LIN {X 0,Y 467.673,Z 382.231,A -85,B 0,C 180,E1 -7731.357,E2 -7731.357} C_VEL
LIN {X 0,Y 467.733,Z 382.223,A -85,B 0,C 180,E1 -7733.963,E2 -7733.963} C_VEL
LIN {X 0,Y 467.851,Z 382.207,A -85,B 0,C 180,E1 -7737.417,E2 -7737.417} C_VEL
LIN {X 0,Y 467.873,Z 382.205,A -85,B 0,C 180,E1 -7740,E2 -7740} C_VEL
LIN {X 0,Y 467.851,Z 382.211,A -85,B 0,C 180,E1 -7742.583,E2 -7742.583} C_VEL
LIN {X 0,Y 467.734,Z 382.223,A -85,B 0,C 180,E1 -7746.038,E2 -7746.038} C_VEL
LIN {X 0,Y 467.674,Z 382.232,A -85,B 0,C 180,E1 -7748.643,E2 -7748.643} C_VEL
LIN {X 0,Y 467.648,Z 382.234,A -85,B 0,C 180,E1 -7752.146,E2 -7752.146} C_VEL
LIN {X 0,Y 467.63,Z 382.235,A -85,B 0,C 180,E1 -7755.695,E2 -7755.695} C_VEL
LIN {X 0,Y 467.609,Z 382.239,A -85,B 0,C 180,E1 -7758.765,E2 -7758.765} C_VEL
LIN {X 0,Y 467.573,Z 382.243,A -85,B 0,C 180,E1 -7761.269,E2 -7761.269} C_VEL
LIN {X 0,Y 467.566,Z 382.246,A -85,B 0,C 180,E1 -7763.944,E2 -7763.944} C_VEL
LIN {X 0,Y 467.621,Z 382.239,A -85,B 0,C 180,E1 -7766.8,E2 -7766.8} C_VEL
LIN {X 0,Y 467.547,Z 382.247,A -85,B 0,C 180,E1 -7769.739,E2 -7769.739} C_VEL
LIN {X 0,Y 467.577,Z 382.243,A -85,B 0,C 180,E1 -7772.759,E2 -7772.759} C_VEL
LIN {X 0,Y 467.552,Z 382.247,A -85,B 0,C 180,E1 -7775.89,E2 -7775.89} C_VEL
LIN {X 0,Y 467.614,Z 382.238,A -85,B 0,C 180,E1 -7779.142,E2 -7779.142} C_VEL
LIN {X 0,Y 467.582,Z 382.243,A -85,B 0,C 180,E1 -7782.568,E2 -7782.568} C_VEL
LIN {X 0,Y 467.566,Z 382.243,A -85,B 0,C 180,E1 -7785.054,E2 -7785.054} C_VEL
LIN {X 0,Y 467.586,Z 382.241,A -85,B 0,C 180,E1 -7787.441,E2 -7787.441} C_VEL
LIN {X 0,Y 467.58,Z 382.242,A -85,B 0,C 180,E1 -7790.856,E2 -7790.856} C_VEL
LIN {X 0,Y 467.561,Z 382.246,A -85,B 0,C 180,E1 -7794.261,E2 -7794.261} C_VEL
LIN {X 0,Y 467.581,Z 382.242,A -85,B 0,C 180,E1 -7797.322,E2 -7797.322} C_VEL
LIN {X 0,Y 467.57,Z 382.243,A -85,B 0,C 180,E1 -7800.668,E2 -7800.668} C_VEL
LIN {X 0,Y 467.617,Z 382.236,A -85,B 0,C 180,E1 -7803.201,E2 -7803.201} C_VEL
LIN {X 0,Y 467.595,Z 382.241,A -85,B 0,C 180,E1 -7806.469,E2 -7806.469} C_VEL
LIN {X 0,Y 467.625,Z 382.238,A -85,B 0,C 180,E1 -7809.778,E2 -7809.778} C_VEL
LIN {X 0,Y 467.609,Z 382.238,A -85,B 0,C 180,E1 -7812.507,E2 -7812.507} C_VEL
LIN {X 0,Y 467.6,Z 382.238,A -85,B 0,C 180,E1 -7815.427,E2 -7815.427} C_VEL
LIN {X 0,Y 466.93,Z 382.324,A -85,B 0,C 180,E1 -7816.146,E2 -7816.146} C_VEL
LIN {X 0,Y 464.086,Z 382.678,A -85,B 0,C 180,E1 -7817.315,E2 -7817.315} C_VEL
LIN {X 0,Y 461.687,Z 382.976,A -85,B 0,C 180,E1 -7818.257,E2 -7818.257} C_VEL
LIN {X 0,Y 460.66,Z 383.103,A -85,B 0,C 180,E1 -7818.984,E2 -7818.984} C_VEL
LIN {X 0,Y 460.578,Z 383.114,A -85,B 0,C 180,E1 -7819.231,E2 -7819.231} C_VEL
LIN {X 0,Y 460.724,Z 383.095,A -85,B 0,C 180,E1 -7822.539,E2 -7822.539} C_VEL
LIN {X 0,Y 460.701,Z 383.098,A -85,B 0,C 180,E1 -7824.749,E2 -7824.749} C_VEL
LIN {X 0,Y 460.642,Z 383.109,A -85,B 0,C 180,E1 -7828.252,E2 -7828.252} C_VEL
LIN {X 0,Y 460.422,Z 383.137,A -85,B 0,C 180,E1 -7830,E2 -7830} C_VEL
LIN {X 0,Y 460.136,Z 383.537,A -85,B 0,C 180,E1 -7830.875,E2 -7830.875} C_VEL
LIN {X 0,Y 460.101,Z 387.168,A -85,B 0,C 180,E1 -7834.38,E2 -7834.38} C_VEL
LIN {X 0,Y 460.05,Z 389.931,A -85,B 0,C 180,E1 -7837.02,E2 -7837.02} C_VEL
LIN {X 0,Y 459.887,Z 393.714,A -85,B 0,C 180,E1 -7840.567,E2 -7840.567} C_VEL
LIN {X 0,Y 459.817,Z 396.601,A -85,B 0,C 180,E1 -7843.254,E2 -7843.254} C_VEL
LIN {X 0,Y 459.747,Z 400.031,A -85,B 0,C 180,E1 -7846.427,E2 -7846.427} C_VEL
LIN {X 0,Y 459.761,Z 400.289,A -85,B 0,C 180,E1 -7846.484,E2 -7846.484} C_VEL
LIN {X 0,Y 463,Z 413.86,A -85,B 0,C 180,E1 -7847.018,E2 -7847.018} C_VEL
LIN {X 0,Y 463.452,Z 417.522,A -85,B 0,C 180,E1 -7847.183,E2 -7847.183} C_VEL
LIN {X 0,Y 462.965,Z 429.882,A -85,B 0,C 180,E1 -7847.788,E2 -7847.788} C_VEL
LIN {X 0,Y 462.562,Z 440.759,A -85,B 0,C 180,E1 -7848.492,E2 -7848.492} C_VEL
LIN {X 0,Y 462.154,Z 450.981,A -85,B 0,C 180,E1 -7849.322,E2 -7849.322} C_VEL
LIN {X 0,Y 461.626,Z 460.435,A -85,B 0,C 180,E1 -7850.264,E2 -7850.264} C_VEL
LIN {X 0,Y 461.106,Z 470.133,A -85,B 0,C 180,E1 -7851.457,E2 -7851.457} C_VEL
LIN {X 0,Y 460.671,Z 478.078,A -85,B 0,C 180,E1 -7852.657,E2 -7852.657} C_VEL
LIN {X 0,Y 460.337,Z 485.075,A -85,B 0,C 180,E1 -7853.959,E2 -7853.959} C_VEL
LIN {X 0,Y 460.054,Z 490.904,A -85,B 0,C 180,E1 -7855.324,E2 -7855.324} C_VEL
LIN {X 0,Y 459.888,Z 495.753,A -85,B 0,C 180,E1 -7856.796,E2 -7856.796} C_VEL
LIN {X 0,Y 459.702,Z 499.35,A -85,B 0,C 180,E1 -7858.29,E2 -7858.29} C_VEL
LIN {X 0,Y 459.602,Z 501.158,A -85,B 0,C 180,E1 -7859.353,E2 -7859.353} C_VEL
LIN {X 0,Y 459.552,Z 502.793,A -85,B 0,C 180,E1 -7861.083,E2 -7861.083} C_VEL
LIN {X 0,Y 459.542,Z 502.954,A -85,B 0,C 180,E1 -7862.739,E2 -7862.739} C_VEL
LIN {X 0,Y 459.603,Z 501.586,A -85,B 0,C 180,E1 -7864.456,E2 -7864.456} C_VEL
LIN {X 0,Y 459.699,Z 499.308,A -85,B 0,C 180,E1 -7865.876,E2 -7865.876} C_VEL
LIN {X 0,Y 459.896,Z 495.681,A -85,B 0,C 180,E1 -7867.377,E2 -7867.377} C_VEL
LIN {X 0,Y 460.107,Z 490.878,A -85,B 0,C 180,E1 -7868.829,E2 -7868.829} C_VEL
LIN {X 0,Y 460.383,Z 484.757,A -85,B 0,C 180,E1 -7870.245,E2 -7870.245} C_VEL
LIN {X 0,Y 460.797,Z 477.118,A -85,B 0,C 180,E1 -7871.639,E2 -7871.639} C_VEL
LIN {X 0,Y 461.249,Z 468.89,A -85,B 0,C 180,E1 -7872.85,E2 -7872.85} C_VEL
LIN {X 0,Y 461.723,Z 459.558,A -85,B 0,C 180,E1 -7873.966,E2 -7873.966} C_VEL
LIN {X 0,Y 462.231,Z 448.885,A -85,B 0,C 180,E1 -7874.991,E2 -7874.991} C_VEL
LIN {X 0,Y 462.725,Z 437.513,A -85,B 0,C 180,E1 -7875.863,E2 -7875.863} C_VEL
LIN {X 0,Y 463.176,Z 425.311,A -85,B 0,C 180,E1 -7876.58,E2 -7876.58} C_VEL
LIN {X 0,Y 463.459,Z 416.793,A -85,B 0,C 180,E1 -7876.969,E2 -7876.969} C_VEL
LIN {X 0,Y 460.901,Z 405.422,A -85,B 0,C 180,E1 -7877.46,E2 -7877.46} C_VEL
LIN {X 0,Y 459.754,Z 400.767,A -85,B 0,C 180,E1 -7877.639,E2 -7877.639} C_VEL
LIN {X 0,Y 459.777,Z 398.225,A -85,B 0,C 180,E1 -7880.059,E2 -7880.059} C_VEL
LIN {X 0,Y 459.846,Z 394.757,A -85,B 0,C 180,E1 -7883.412,E2 -7883.412} C_VEL
LIN {X 0,Y 459.973,Z 391.444,A -85,B 0,C 180,E1 -7886.629,E2 -7886.629} C_VEL
LIN {X 0,Y 460.058,Z 388.286,A -85,B 0,C 180,E1 -7889.727,E2 -7889.727} C_VEL
LIN {X 0,Y 460.11,Z 385.256,A -85,B 0,C 180,E1 -7892.726,E2 -7892.726} C_VEL
LIN {X 0,Y 460.168,Z 383.268,A -85,B 0,C 180,E1 -7894.682,E2 -7894.682} C_VEL
LIN {X 0,Y 460.464,Z 383.133,A -85,B 0,C 180,E1 -7897.569,E2 -7897.569} C_VEL
LIN {X 0,Y 460.565,Z 383.117,A -85,B 0,C 180,E1 -7900.384,E2 -7900.384} C_VEL
LIN {X 0,Y 460.56,Z 383.118,A -85,B 0,C 180,E1 -7903.146,E2 -7903.146} C_VEL
LIN {X 0,Y 460.549,Z 383.121,A -85,B 0,C 180,E1 -7905.868,E2 -7905.868} C_VEL
LIN {X 0,Y 460.607,Z 383.111,A -85,B 0,C 180,E1 -7908.559,E2 -7908.559} C_VEL
LIN {X 0,Y 460.689,Z 383.1,A -85,B 0,C 180,E1 -7912.108,E2 -7912.108} C_VEL
LIN {X 0,Y 460.691,Z 383.099,A -85,B 0,C 180,E1 -7914.748,E2 -7914.748} C_VEL
LIN {X 0,Y 460.819,Z 383.082,A -85,B 0,C 180,E1 -7917.378,E2 -7917.378} C_VEL
LIN {X 0,Y 460.846,Z 383.08,A -85,B 0,C 180,E1 -7920,E2 -7920} C_VEL
LIN {X 0,Y 460.818,Z 383.084,A -85,B 0,C 180,E1 -7922.622,E2 -7922.622} C_VEL
LIN {X 0,Y 460.703,Z 383.099,A -85,B 0,C 180,E1 -7926.13,E2 -7926.13} C_VEL
LIN {X 0,Y 460.623,Z 383.11,A -85,B 0,C 180,E1 -7928.776,E2 -7928.776} C_VEL
LIN {X 0,Y 460.607,Z 383.112,A -85,B 0,C 180,E1 -7932.445,E2 -7932.445} C_VEL
LIN {X 0,Y 460.594,Z 383.112,A -85,B 0,C 180,E1 -7935.998,E2 -7935.998} C_VEL
LIN {X 0,Y 460.565,Z 383.114,A -85,B 0,C 180,E1 -7938.902,E2 -7938.902} C_VEL
LIN {X 0,Y 460.51,Z 383.123,A -85,B 0,C 180,E1 -7941.486,E2 -7941.486} C_VEL
LIN {X 0,Y 460.537,Z 383.121,A -85,B 0,C 180,E1 -7944.333,E2 -7944.333} C_VEL
LIN {X 0,Y 460.579,Z 383.116,A -85,B 0,C 180,E1 -7947.243,E2 -7947.243} C_VEL
LIN {X 0,Y 460.505,Z 383.125,A -85,B 0,C 180,E1 -7950.24,E2 -7950.24} C_VEL
LIN {X 0,Y 460.515,Z 383.125,A -85,B 0,C 180,E1 -7953.326,E2 -7953.326} C_VEL
LIN {X 0,Y 460.473,Z 383.132,A -85,B 0,C 180,E1 -7956.53,E2 -7956.53} C_VEL
LIN {X 0,Y 460.575,Z 383.117,A -85,B 0,C 180,E1 -7959.858,E2 -7959.858} C_VEL
LIN {X 0,Y 460.51,Z 383.124,A -85,B 0,C 180,E1 -7962.901,E2 -7962.901} C_VEL
LIN {X 0,Y 460.509,Z 383.125,A -85,B 0,C 180,E1 -7965.831,E2 -7965.831} C_VEL
LIN {X 0,Y 460.581,Z 383.262,A -85,B 0,C 180,E1 -7968.847,E2 -7968.847} C_VEL
LIN {X 0,Y 461.978,Z 390.924,A -85,B 0,C 180,E1 -7972.519,E2 -7972.519} C_VEL
LIN {X 0,Y 462.403,Z 394.851,A -85,B 0,C 180,E1 -7974.202,E2 -7974.202} C_VEL
LIN {X 0,Y 462.054,Z 401.187,A -85,B 0,C 180,E1 -7976.8,E2 -7976.8} C_VEL
LIN {X 0,Y 461.502,Z 410.096,A -85,B 0,C 180,E1 -7980.23,E2 -7980.23} C_VEL
LIN {X 0,Y 461.151,Z 418.397,A -85,B 0,C 180,E1 -7983.283,E2 -7983.283} C_VEL
LIN {X 0,Y 460.78,Z 427.79,A -85,B 0,C 180,E1 -7986.637,E2 -7986.637} C_VEL
LIN {X 0,Y 460.497,Z 437.508,A -85,B 0,C 180,E1 -7989.917,E2 -7989.917} C_VEL
LIN {X 0,Y 460.237,Z 445.764,A -85,B 0,C 180,E1 -7992.676,E2 -7992.676} C_VEL
LIN {X 0,Y 460.163,Z 450.69,A -85,B 0,C 180,E1 -7994.339,E2 -7994.339} C_VEL
LIN {X 0,Y 462.544,Z 465.256,A -85,B 0,C 180,E1 -7994.813,E2 -7994.813} C_VEL
LIN {X 0,Y 463.237,Z 471.072,A -85,B 0,C 180,E1 -7995.054,E2 -7995.054} C_VEL
LIN {X 0,Y 462.854,Z 482.753,A -85,B 0,C 180,E1 -7995.603,E2 -7995.603} C_VEL
LIN {X 0,Y 462.294,Z 495.103,A -85,B 0,C 180,E1 -7996.371,E2 -7996.371} C_VEL
LIN {X 0,Y 461.859,Z 505.182,A -85,B 0,C 180,E1 -7997.168,E2 -7997.168} C_VEL
LIN {X 0,Y 461.401,Z 515.131,A -85,B 0,C 180,E1 -7998.134,E2 -7998.134} C_VEL
LIN {X 0,Y 460.835,Z 524.354,A -85,B 0,C 180,E1 -7999.233,E2 -7999.233} C_VEL
LIN {X 0,Y 460.396,Z 533.354,A -85,B 0,C 180,E1 -8000.555,E2 -8000.555} C_VEL
LIN {X 0,Y 460.054,Z 540.602,A -85,B 0,C 180,E1 -8001.876,E2 -8001.876} C_VEL
LIN {X 0,Y 459.848,Z 545.496,A -85,B 0,C 180,E1 -8002.977,E2 -8002.977} C_VEL
LIN {X 0,Y 459.756,Z 550.26,A -85,B 0,C 180,E1 -8004.297,E2 -8004.297} C_VEL
LIN {X 0,Y 459.58,Z 553.894,A -85,B 0,C 180,E1 -8005.615,E2 -8005.615} C_VEL
LIN {X 0,Y 459.591,Z 555.773,A -85,B 0,C 180,E1 -8006.493,E2 -8006.493} C_VEL
LIN {X 0,Y 459.57,Z 557.175,A -85,B 0,C 180,E1 -8007.37,E2 -8007.37} C_VEL
LIN {X 0,Y 459.494,Z 558.779,A -85,B 0,C 180,E1 -8009.123,E2 -8009.123} C_VEL
LIN {X 0,Y 459.474,Z 558.994,A -85,B 0,C 180,E1 -8010,E2 -8010} C_VEL
LIN {X 0,Y 459.494,Z 558.779,A -85,B 0,C 180,E1 -8010.876,E2 -8010.876} C_VEL
LIN {X 0,Y 459.57,Z 557.179,A -85,B 0,C 180,E1 -8012.629,E2 -8012.629} C_VEL
LIN {X 0,Y 459.591,Z 555.777,A -85,B 0,C 180,E1 -8013.507,E2 -8013.507} C_VEL
LIN {X 0,Y 459.634,Z 552.819,A -85,B 0,C 180,E1 -8014.824,E2 -8014.824} C_VEL
LIN {X 0,Y 459.757,Z 548.818,A -85,B 0,C 180,E1 -8016.142,E2 -8016.142} C_VEL
LIN {X 0,Y 459.929,Z 542.664,A -85,B 0,C 180,E1 -8017.683,E2 -8017.683} C_VEL
LIN {X 0,Y 460.287,Z 535.951,A -85,B 0,C 180,E1 -8019.004,E2 -8019.004} C_VEL
LIN {X 0,Y 460.699,Z 527.624,A -85,B 0,C 180,E1 -8020.325,E2 -8020.325} C_VEL
LIN {X 0,Y 461.15,Z 519.095,A -85,B 0,C 180,E1 -8021.427,E2 -8021.427} C_VEL
LIN {X 0,Y 461.664,Z 508.859,A -85,B 0,C 180,E1 -8022.5,E2 -8022.5} C_VEL
LIN {X 0,Y 462.174,Z 496.862,A -85,B 0,C 180,E1 -8023.509,E2 -8023.509} C_VEL
LIN {X 0,Y 462.717,Z 484.815,A -85,B 0,C 180,E1 -8024.289,E2 -8024.289} C_VEL
LIN {X 0,Y 463.22,Z 472.452,A -85,B 0,C 180,E1 -8024.89,E2 -8024.89} C_VEL
LIN {X 0,Y 463.011,Z 468.654,A -85,B 0,C 180,E1 -8025.05,E2 -8025.05} C_VEL
LIN {X 0,Y 460.929,Z 455.877,A -85,B 0,C 180,E1 -8025.515,E2 -8025.515} C_VEL
LIN {X 0,Y 460.169,Z 450.853,A -85,B 0,C 180,E1 -8025.661,E2 -8025.661} C_VEL
LIN {X 0,Y 460.459,Z 440.42,A -85,B 0,C 180,E1 -8029.178,E2 -8029.178} C_VEL
LIN {X 0,Y 460.726,Z 430.867,A -85,B 0,C 180,E1 -8032.417,E2 -8032.417} C_VEL
LIN {X 0,Y 460.993,Z 422.694,A -85,B 0,C 180,E1 -8035.268,E2 -8035.268} C_VEL
LIN {X 0,Y 461.385,Z 414.794,A -85,B 0,C 180,E1 -8038.177,E2 -8038.177} C_VEL
LIN {X 0,Y 461.803,Z 405.886,A -85,B 0,C 180,E1 -8041.543,E2 -8041.543} C_VEL
LIN {X 0,Y 462.222,Z 399.011,A -85,B 0,C 180,E1 -8044.233,E2 -8044.233} C_VEL
LIN {X 0,Y 462.401,Z 393.857,A -85,B 0,C 180,E1 -8046.337,E2 -8046.337} C_VEL
LIN {X 0,Y 461.392,Z 387.782,A -85,B 0,C 180,E1 -8049.028,E2 -8049.028} C_VEL
LIN {X 0,Y 460.548,Z 383.118,A -85,B 0,C 180,E1 -8051.303,E2 -8051.303} C_VEL
LIN {X 0,Y 460.512,Z 383.124,A -85,B 0,C 180,E1 -8054.588,E2 -8054.588} C_VEL
LIN {X 0,Y 460.519,Z 383.122,A -85,B 0,C 180,E1 -8057.818,E2 -8057.818} C_VEL
LIN {X 0,Y 460.562,Z 383.118,A -85,B 0,C 180,E1 -8061.098,E2 -8061.098} C_VEL
LIN {X 0,Y 460.507,Z 383.124,A -85,B 0,C 180,E1 -8064.554,E2 -8064.554} C_VEL
LIN {X 0,Y 460.525,Z 383.119,A -85,B 0,C 180,E1 -8067.715,E2 -8067.715} C_VEL
LIN {X 0,Y 460.532,Z 383.122,A -85,B 0,C 180,E1 -8070.768,E2 -8070.768} C_VEL
LIN {X 0,Y 460.56,Z 383.116,A -85,B 0,C 180,E1 -8073.735,E2 -8073.735} C_VEL
LIN {X 0,Y 460.538,Z 383.121,A -85,B 0,C 180,E1 -8076.624,E2 -8076.624} C_VEL
LIN {X 0,Y 460.544,Z 383.119,A -85,B 0,C 180,E1 -8079.452,E2 -8079.452} C_VEL
LIN {X 0,Y 460.551,Z 383.118,A -85,B 0,C 180,E1 -8082.23,E2 -8082.23} C_VEL
LIN {X 0,Y 460.556,Z 383.119,A -85,B 0,C 180,E1 -8084.965,E2 -8084.965} C_VEL
LIN {X 0,Y 460.604,Z 383.113,A -85,B 0,C 180,E1 -8088.559,E2 -8088.559} C_VEL
LIN {X 0,Y 460.686,Z 383.101,A -85,B 0,C 180,E1 -8092.108,E2 -8092.108} C_VEL
LIN {X 0,Y 460.688,Z 383.103,A -85,B 0,C 180,E1 -8094.748,E2 -8094.748} C_VEL
LIN {X 0,Y 460.816,Z 383.084,A -85,B 0,C 180,E1 -8097.378,E2 -8097.378} C_VEL
LIN {X 0,Y 460.844,Z 383.081,A -85,B 0,C 180,E1 -8100,E2 -8100} C_VEL
LIN {X 0,Y 460.816,Z 383.087,A -85,B 0,C 180,E1 -8102.623,E2 -8102.623} C_VEL
LIN {X 0,Y 460.701,Z 383.1,A -85,B 0,C 180,E1 -8106.13,E2 -8106.13} C_VEL
LIN {X 0,Y 460.621,Z 383.11,A -85,B 0,C 180,E1 -8108.776,E2 -8108.776} C_VEL
LIN {X 0,Y 460.604,Z 383.113,A -85,B 0,C 180,E1 -8112.445,E2 -8112.445} C_VEL
LIN {X 0,Y 460.591,Z 383.113,A -85,B 0,C 180,E1 -8115.998,E2 -8115.998} C_VEL
LIN {X 0,Y 460.563,Z 383.117,A -85,B 0,C 180,E1 -8118.902,E2 -8118.902} C_VEL
LIN {X 0,Y 460.508,Z 383.122,A -85,B 0,C 180,E1 -8121.486,E2 -8121.486} C_VEL
LIN {X 0,Y 460.535,Z 383.121,A -85,B 0,C 180,E1 -8124.333,E2 -8124.333} C_VEL
LIN {X 0,Y 460.577,Z 383.114,A -85,B 0,C 180,E1 -8127.244,E2 -8127.244} C_VEL
LIN {X 0,Y 460.504,Z 383.126,A -85,B 0,C 180,E1 -8130.241,E2 -8130.241} C_VEL
LIN {X 0,Y 460.523,Z 383.12,A -85,B 0,C 180,E1 -8133.326,E2 -8133.326} C_VEL
LIN {X 0,Y 460.475,Z 383.128,A -85,B 0,C 180,E1 -8136.53,E2 -8136.53} C_VEL
LIN {X 0,Y 460.573,Z 383.116,A -85,B 0,C 180,E1 -8139.858,E2 -8139.858} C_VEL
LIN {X 0,Y 460.509,Z 383.122,A -85,B 0,C 180,E1 -8142.901,E2 -8142.901} C_VEL
LIN {X 0,Y 460.508,Z 383.124,A -85,B 0,C 180,E1 -8145.831,E2 -8145.831} C_VEL
LIN {X 0,Y 460.528,Z 383.12,A -85,B 0,C 180,E1 -8148.99,E2 -8148.99} C_VEL
LIN {X 0,Y 460.524,Z 383.12,A -85,B 0,C 180,E1 -8151.268,E2 -8151.268} C_VEL
LIN {X 0,Y 460.511,Z 383.124,A -85,B 0,C 180,E1 -8154.556,E2 -8154.556} C_VEL
LIN {X 0,Y 460.531,Z 383.121,A -85,B 0,C 180,E1 -8157.717,E2 -8157.717} C_VEL
LIN {X 0,Y 460.54,Z 383.118,A -85,B 0,C 180,E1 -8160.77,E2 -8160.77} C_VEL
LIN {X 0,Y 460.564,Z 383.119,A -85,B 0,C 180,E1 -8163.736,E2 -8163.736} C_VEL
LIN {X 0,Y 460.548,Z 383.118,A -85,B 0,C 180,E1 -8166.625,E2 -8166.625} C_VEL
LIN {X 0,Y 460.554,Z 383.119,A -85,B 0,C 180,E1 -8169.454,E2 -8169.454} C_VEL
LIN {X 0,Y 460.56,Z 383.119,A -85,B 0,C 180,E1 -8172.231,E2 -8172.231} C_VEL
LIN {X 0,Y 460.568,Z 383.115,A -85,B 0,C 180,E1 -8174.965,E2 -8174.965} C_VEL
LIN {X 0,Y 460.614,Z 383.11,A -85,B 0,C 180,E1 -8178.56,E2 -8178.56} C_VEL
LIN {X 0,Y 460.578,Z 383.114,A -85,B 0,C 180,E1 -8179.231,E2 -8179.231} C_VEL
LIN {X 0,Y 459.922,Z 383.199,A -85,B 0,C 180,E1 -8179.961,E2 -8179.961} C_VEL
LIN {X 0,Y 457.106,Z 383.549,A -85,B 0,C 180,E1 -8181.147,E2 -8181.147} C_VEL
LIN {X 0,Y 454.729,Z 383.845,A -85,B 0,C 180,E1 -8182.105,E2 -8182.105} C_VEL
LIN {X 0,Y 453.718,Z 383.967,A -85,B 0,C 180,E1 -8182.844,E2 -8182.844} C_VEL
LIN {X 0,Y 453.641,Z 383.976,A -85,B 0,C 180,E1 -8183.094,E2 -8183.094} C_VEL
LIN {X 0,Y 453.675,Z 383.973,A -85,B 0,C 180,E1 -8184.667,E2 -8184.667} C_VEL
LIN {X 0,Y 453.615,Z 383.985,A -85,B 0,C 180,E1 -8188.225,E2 -8188.225} C_VEL
LIN {X 0,Y 453.392,Z 384.013,A -85,B 0,C 180,E1 -8190,E2 -8190} C_VEL
LIN {X 0,Y 453.068,Z 384.308,A -85,B 0,C 180,E1 -8190.889,E2 -8190.889} C_VEL
LIN {X 0,Y 453.038,Z 387.969,A -85,B 0,C 180,E1 -8194.449,E2 -8194.449} C_VEL
LIN {X 0,Y 452.964,Z 390.73,A -85,B 0,C 180,E1 -8197.13,E2 -8197.13} C_VEL
LIN {X 0,Y 452.838,Z 394.587,A -85,B 0,C 180,E1 -8200.733,E2 -8200.733} C_VEL
LIN {X 0,Y 452.733,Z 397.492,A -85,B 0,C 180,E1 -8203.465,E2 -8203.465} C_VEL
LIN {X 0,Y 452.696,Z 400.503,A -85,B 0,C 180,E1 -8206.227,E2 -8206.227} C_VEL
LIN {X 0,Y 456.108,Z 414.964,A -85,B 0,C 180,E1 -8206.817,E2 -8206.817} C_VEL
LIN {X 0,Y 456.603,Z 417.501,A -85,B 0,C 180,E1 -8206.941,E2 -8206.941} C_VEL
LIN {X 0,Y 456.094,Z 430.76,A -85,B 0,C 180,E1 -8207.602,E2 -8207.602} C_VEL
LIN {X 0,Y 455.647,Z 441.569,A -85,B 0,C 180,E1 -8208.316,E2 -8208.316} C_VEL
LIN {X 0,Y 455.136,Z 452.929,A -85,B 0,C 180,E1 -8209.276,E2 -8209.276} C_VEL
LIN {X 0,Y 454.533,Z 463.217,A -85,B 0,C 180,E1 -8210.358,E2 -8210.358} C_VEL
LIN {X 0,Y 454.005,Z 472.929,A -85,B 0,C 180,E1 -8211.635,E2 -8211.635} C_VEL
LIN {X 0,Y 453.499,Z 481.425,A -85,B 0,C 180,E1 -8213.036,E2 -8213.036} C_VEL
LIN {X 0,Y 453.161,Z 488.507,A -85,B 0,C 180,E1 -8214.51,E2 -8214.51} C_VEL
LIN {X 0,Y 452.895,Z 493.503,A -85,B 0,C 180,E1 -8215.836,E2 -8215.836} C_VEL
LIN {X 0,Y 452.794,Z 497.6,A -85,B 0,C 180,E1 -8217.25,E2 -8217.25} C_VEL
LIN {X 0,Y 452.572,Z 500.759,A -85,B 0,C 180,E1 -8218.776,E2 -8218.776} C_VEL
LIN {X 0,Y 452.497,Z 502.208,A -85,B 0,C 180,E1 -8219.802,E2 -8219.802} C_VEL
LIN {X 0,Y 452.461,Z 503.357,A -85,B 0,C 180,E1 -8221.316,E2 -8221.316} C_VEL
LIN {X 0,Y 452.471,Z 503.272,A -85,B 0,C 180,E1 -8222.991,E2 -8222.991} C_VEL
LIN {X 0,Y 452.525,Z 501.894,A -85,B 0,C 180,E1 -8224.601,E2 -8224.601} C_VEL
LIN {X 0,Y 452.661,Z 499.306,A -85,B 0,C 180,E1 -8226.162,E2 -8226.162} C_VEL
LIN {X 0,Y 452.869,Z 495.523,A -85,B 0,C 180,E1 -8227.677,E2 -8227.677} C_VEL
LIN {X 0,Y 453.12,Z 490.496,A -85,B 0,C 180,E1 -8229.148,E2 -8229.148} C_VEL
LIN {X 0,Y 453.472,Z 484.031,A -85,B 0,C 180,E1 -8230.611,E2 -8230.611} C_VEL
LIN {X 0,Y 453.879,Z 476.356,A -85,B 0,C 180,E1 -8231.991,E2 -8231.991} C_VEL
LIN {X 0,Y 454.33,Z 468.446,A -85,B 0,C 180,E1 -8233.139,E2 -8233.139} C_VEL
LIN {X 0,Y 454.873,Z 458.449,A -85,B 0,C 180,E1 -8234.315,E2 -8234.315} C_VEL
LIN {X 0,Y 455.35,Z 448.873,A -85,B 0,C 180,E1 -8235.232,E2 -8235.232} C_VEL
LIN {X 0,Y 455.862,Z 438.031,A -85,B 0,C 180,E1 -8236.071,E2 -8236.071} C_VEL
LIN {X 0,Y 456.32,Z 426.219,A -85,B 0,C 180,E1 -8236.781,E2 -8236.781} C_VEL
LIN {X 0,Y 456.459,Z 416.694,A -85,B 0,C 180,E1 -8237.229,E2 -8237.229} C_VEL
LIN {X 0,Y 453.32,Z 403.86,A -85,B 0,C 180,E1 -8237.78,E2 -8237.78} C_VEL
LIN {X 0,Y 452.684,Z 401.216,A -85,B 0,C 180,E1 -8237.894,E2 -8237.894} C_VEL
LIN {X 0,Y 452.71,Z 398.088,A -85,B 0,C 180,E1 -8240.914,E2 -8240.914} C_VEL
LIN {X 0,Y 452.808,Z 395.044,A -85,B 0,C 180,E1 -8243.857,E2 -8243.857} C_VEL
LIN {X 0,Y 452.929,Z 391.77,A -85,B 0,C 180,E1 -8247.106,E2 -8247.106} C_VEL
LIN {X 0,Y 453.009,Z 388.584,A -85,B 0,C 180,E1 -8250.234,E2 -8250.234} C_VEL
LIN {X 0,Y 453.064,Z 385.546,A -85,B 0,C 180,E1 -8253.266,E2 -8253.266} C_VEL
LIN {X 0,Y 453.127,Z 384.547,A -85,B 0,C 180,E1 -8254.26,E2 -8254.26} C_VEL
LIN {X 0,Y 453.189,Z 384.038,A -85,B 0,C 180,E1 -8255.246,E2 -8255.246} C_VEL
LIN {X 0,Y 453.459,Z 384.006,A -85,B 0,C 180,E1 -8258.163,E2 -8258.163} C_VEL
LIN {X 0,Y 453.517,Z 383.997,A -85,B 0,C 180,E1 -8261.008,E2 -8261.008} C_VEL
LIN {X 0,Y 453.563,Z 383.988,A -85,B 0,C 180,E1 -8263.879,E2 -8263.879} C_VEL
LIN {X 0,Y 453.558,Z 383.99,A -85,B 0,C 180,E1 -8267.471,E2 -8267.471} C_VEL
LIN {X 0,Y 453.587,Z 383.986,A -85,B 0,C 180,E1 -8271.086,E2 -8271.086} C_VEL
LIN {X 0,Y 453.671,Z 383.975,A -85,B 0,C 180,E1 -8273.774,E2 -8273.774} C_VEL
LIN {X 0,Y 453.759,Z 383.962,A -85,B 0,C 180,E1 -8277.337,E2 -8277.337} C_VEL
LIN {X 0,Y 453.816,Z 383.955,A -85,B 0,C 180,E1 -8280,E2 -8280} C_VEL
LIN {X 0,Y 453.759,Z 383.964,A -85,B 0,C 180,E1 -8282.663,E2 -8282.663} C_VEL
LIN {X 0,Y 453.67,Z 383.976,A -85,B 0,C 180,E1 -8286.225,E2 -8286.225} C_VEL
LIN {X 0,Y 453.587,Z 383.987,A -85,B 0,C 180,E1 -8288.913,E2 -8288.913} C_VEL
LIN {X 0,Y 453.557,Z 383.99,A -85,B 0,C 180,E1 -8292.529,E2 -8292.529} C_VEL
LIN {X 0,Y 453.539,Z 383.99,A -85,B 0,C 180,E1 -8296.196,E2 -8296.196} C_VEL
LIN {X 0,Y 453.514,Z 383.992,A -85,B 0,C 180,E1 -8299.041,E2 -8299.041} C_VEL
LIN {X 0,Y 453.471,Z 384.001,A -85,B 0,C 180,E1 -8301.836,E2 -8301.836} C_VEL
LIN {X 0,Y 453.509,Z 383.997,A -85,B 0,C 180,E1 -8304.735,E2 -8304.735} C_VEL
LIN {X 0,Y 453.533,Z 383.994,A -85,B 0,C 180,E1 -8307.961,E2 -8307.961} C_VEL
LIN {X 0,Y 453.46,Z 384.002,A -85,B 0,C 180,E1 -8311.525,E2 -8311.525} C_VEL
LIN {X 0,Y 453.478,Z 384.001,A -85,B 0,C 180,E1 -8314.777,E2 -8314.777} C_VEL
LIN {X 0,Y 453.482,Z 384,A -85,B 0,C 180,E1 -8318.31,E2 -8318.31} C_VEL
LIN {X 0,Y 453.513,Z 383.997,A -85,B 0,C 180,E1 -8320.607,E2 -8320.607} C_VEL
LIN {X 0,Y 453.463,Z 384.002,A -85,B 0,C 180,E1 -8324.221,E2 -8324.221} C_VEL
LIN {X 0,Y 453.461,Z 384.004,A -85,B 0,C 180,E1 -8327.006,E2 -8327.006} C_VEL
LIN {X 0,Y 453.526,Z 384.139,A -85,B 0,C 180,E1 -8328.513,E2 -8328.513} C_VEL
LIN {X 0,Y 454.528,Z 389.726,A -85,B 0,C 180,E1 -8331.25,E2 -8331.25} C_VEL
LIN {X 0,Y 455.317,Z 394.234,A -85,B 0,C 180,E1 -8333.383,E2 -8333.383} C_VEL
LIN {X 0,Y 455.279,Z 398.473,A -85,B 0,C 180,E1 -8335.17,E2 -8335.17} C_VEL
LIN {X 0,Y 454.88,Z 404.896,A -85,B 0,C 180,E1 -8337.787,E2 -8337.787} C_VEL
LIN {X 0,Y 454.363,Z 414.1,A -85,B 0,C 180,E1 -8341.347,E2 -8341.347} C_VEL
LIN {X 0,Y 453.945,Z 422.089,A -85,B 0,C 180,E1 -8344.311,E2 -8344.311} C_VEL
LIN {X 0,Y 453.673,Z 430.213,A -85,B 0,C 180,E1 -8347.215,E2 -8347.215} C_VEL
LIN {X 0,Y 453.409,Z 439.867,A -85,B 0,C 180,E1 -8350.534,E2 -8350.534} C_VEL
LIN {X 0,Y 453.075,Z 450.258,A -85,B 0,C 180,E1 -8354.098,E2 -8354.098} C_VEL
LIN {X 0,Y 455.051,Z 462.267,A -85,B 0,C 180,E1 -8354.475,E2 -8354.475} C_VEL
LIN {X 0,Y 456.336,Z 471.909,A -85,B 0,C 180,E1 -8354.879,E2 -8354.879} C_VEL
LIN {X 0,Y 455.861,Z 484.275,A -85,B 0,C 180,E1 -8355.491,E2 -8355.491} C_VEL
LIN {X 0,Y 455.282,Z 496.181,A -85,B 0,C 180,E1 -8356.271,E2 -8356.271} C_VEL
LIN {X 0,Y 454.791,Z 506.767,A -85,B 0,C 180,E1 -8357.156,E2 -8357.156} C_VEL
LIN {X 0,Y 454.295,Z 516.635,A -85,B 0,C 180,E1 -8358.172,E2 -8358.172} C_VEL
LIN {X 0,Y 453.714,Z 525.536,A -85,B 0,C 180,E1 -8359.288,E2 -8359.288} C_VEL
LIN {X 0,Y 453.299,Z 534.234,A -85,B 0,C 180,E1 -8360.631,E2 -8360.631} C_VEL
LIN {X 0,Y 452.924,Z 541.184,A -85,B 0,C 180,E1 -8361.972,E2 -8361.972} C_VEL
LIN {X 0,Y 452.71,Z 547.416,A -85,B 0,C 180,E1 -8363.493,E2 -8363.493} C_VEL
LIN {X 0,Y 452.567,Z 552.377,A -85,B 0,C 180,E1 -8365.1,E2 -8365.1} C_VEL
LIN {X 0,Y 452.494,Z 555.337,A -85,B 0,C 180,E1 -8366.438,E2 -8366.438} C_VEL
LIN {X 0,Y 452.496,Z 556.749,A -85,B 0,C 180,E1 -8367.329,E2 -8367.329} C_VEL
LIN {X 0,Y 452.433,Z 558.367,A -85,B 0,C 180,E1 -8369.11,E2 -8369.11} C_VEL
LIN {X 0,Y 452.41,Z 558.586,A -85,B 0,C 180,E1 -8370,E2 -8370} C_VEL
LIN {X 0,Y 452.433,Z 558.371,A -85,B 0,C 180,E1 -8370.89,E2 -8370.89} C_VEL
LIN {X 0,Y 452.496,Z 556.759,A -85,B 0,C 180,E1 -8372.67,E2 -8372.67} C_VEL
LIN {X 0,Y 452.493,Z 555.351,A -85,B 0,C 180,E1 -8373.562,E2 -8373.562} C_VEL
LIN {X 0,Y 452.567,Z 552.394,A -85,B 0,C 180,E1 -8374.899,E2 -8374.899} C_VEL
LIN {X 0,Y 452.686,Z 547.533,A -85,B 0,C 180,E1 -8376.481,E2 -8376.481} C_VEL
LIN {X 0,Y 452.926,Z 541.219,A -85,B 0,C 180,E1 -8378.027,E2 -8378.027} C_VEL
LIN {X 0,Y 453.309,Z 534.281,A -85,B 0,C 180,E1 -8379.368,E2 -8379.368} C_VEL
LIN {X 0,Y 453.697,Z 525.596,A -85,B 0,C 180,E1 -8380.712,E2 -8380.712} C_VEL
LIN {X 0,Y 454.277,Z 516.707,A -85,B 0,C 180,E1 -8381.828,E2 -8381.828} C_VEL
LIN {X 0,Y 454.807,Z 506.763,A -85,B 0,C 180,E1 -8382.852,E2 -8382.852} C_VEL
LIN {X 0,Y 455.266,Z 496.288,A -85,B 0,C 180,E1 -8383.729,E2 -8383.729} C_VEL
LIN {X 0,Y 455.803,Z 484.386,A -85,B 0,C 180,E1 -8384.51,E2 -8384.51} C_VEL
LIN {X 0,Y 456.338,Z 472.025,A -85,B 0,C 180,E1 -8385.12,E2 -8385.12} C_VEL
LIN {X 0,Y 454.636,Z 459.724,A -85,B 0,C 180,E1 -8385.622,E2 -8385.622} C_VEL
LIN {X 0,Y 453.075,Z 450.464,A -85,B 0,C 180,E1 -8385.902,E2 -8385.902} C_VEL
LIN {X 0,Y 453.416,Z 440.196,A -85,B 0,C 180,E1 -8389.466,E2 -8389.466} C_VEL
LIN {X 0,Y 453.651,Z 431.951,A -85,B 0,C 180,E1 -8392.305,E2 -8392.305} C_VEL
LIN {X 0,Y 453.951,Z 423.813,A -85,B 0,C 180,E1 -8395.197,E2 -8395.197} C_VEL
LIN {X 0,Y 454.363,Z 415.899,A -85,B 0,C 180,E1 -8398.156,E2 -8398.156} C_VEL
LIN {X 0,Y 454.844,Z 406.396,A -85,B 0,C 180,E1 -8401.806,E2 -8401.806} C_VEL
LIN {X 0,Y 455.256,Z 400.132,A -85,B 0,C 180,E1 -8404.295,E2 -8404.295} C_VEL
LIN {X 0,Y 455.481,Z 396.271,A -85,B 0,C 180,E1 -8405.896,E2 -8405.896} C_VEL
LIN {X 0,Y 454.877,Z 391.457,A -85,B 0,C 180,E1 -8408.004,E2 -8408.004} C_VEL
LIN {X 0,Y 453.518,Z 384.02,A -85,B 0,C 180,E1 -8411.506,E2 -8411.506} C_VEL
LIN {X 0,Y 453.482,Z 383.999,A -85,B 0,C 180,E1 -8414.528,E2 -8414.528} C_VEL
LIN {X 0,Y 453.476,Z 384,A -85,B 0,C 180,E1 -8418.209,E2 -8418.209} C_VEL
LIN {X 0,Y 453.526,Z 383.995,A -85,B 0,C 180,E1 -8420.787,E2 -8420.787} C_VEL
LIN {X 0,Y 453.451,Z 384.001,A -85,B 0,C 180,E1 -8423.917,E2 -8423.917} C_VEL
LIN {X 0,Y 453.476,Z 384.001,A -85,B 0,C 180,E1 -8427.151,E2 -8427.151} C_VEL
LIN {X 0,Y 453.468,Z 383.999,A -85,B 0,C 180,E1 -8430.268,E2 -8430.268} C_VEL
LIN {X 0,Y 453.506,Z 383.996,A -85,B 0,C 180,E1 -8433.294,E2 -8433.294} C_VEL
LIN {X 0,Y 453.495,Z 383.997,A -85,B 0,C 180,E1 -8436.238,E2 -8436.238} C_VEL
LIN {X 0,Y 453.475,Z 384.001,A -85,B 0,C 180,E1 -8439.117,E2 -8439.117} C_VEL
LIN {X 0,Y 453.503,Z 383.995,A -85,B 0,C 180,E1 -8441.944,E2 -8441.944} C_VEL
LIN {X 0,Y 453.53,Z 383.994,A -85,B 0,C 180,E1 -8444.726,E2 -8444.726} C_VEL
LIN {X 0,Y 453.552,Z 383.991,A -85,B 0,C 180,E1 -8448.379,E2 -8448.379} C_VEL
LIN {X 0,Y 453.643,Z 383.978,A -85,B 0,C 180,E1 -8451.985,E2 -8451.985} C_VEL
LIN {X 0,Y 453.662,Z 383.978,A -85,B 0,C 180,E1 -8454.667,E2 -8454.667} C_VEL
LIN {X 0,Y 453.756,Z 383.963,A -85,B 0,C 180,E1 -8457.337,E2 -8457.337} C_VEL
LIN {X 0,Y 453.814,Z 383.957,A -85,B 0,C 180,E1 -8460,E2 -8460} C_VEL
LIN {X 0,Y 453.757,Z 383.967,A -85,B 0,C 180,E1 -8462.663,E2 -8462.663} C_VEL
LIN {X 0,Y 453.668,Z 383.977,A -85,B 0,C 180,E1 -8466.226,E2 -8466.226} C_VEL
LIN {X 0,Y 453.585,Z 383.987,A -85,B 0,C 180,E1 -8468.914,E2 -8468.914} C_VEL
LIN {X 0,Y 453.554,Z 383.992,A -85,B 0,C 180,E1 -8472.529,E2 -8472.529} C_VEL
LIN {X 0,Y 453.536,Z 383.994,A -85,B 0,C 180,E1 -8476.196,E2 -8476.196} C_VEL
LIN {X 0,Y 453.512,Z 383.995,A -85,B 0,C 180,E1 -8479.041,E2 -8479.041} C_VEL
LIN {X 0,Y 453.469,Z 384.001,A -85,B 0,C 180,E1 -8481.837,E2 -8481.837} C_VEL
LIN {X 0,Y 453.507,Z 383.996,A -85,B 0,C 180,E1 -8484.735,E2 -8484.735} C_VEL
LIN {X 0,Y 453.53,Z 383.993,A -85,B 0,C 180,E1 -8487.962,E2 -8487.962} C_VEL
LIN {X 0,Y 453.46,Z 384,A -85,B 0,C 180,E1 -8491.526,E2 -8491.526} C_VEL
LIN {X 0,Y 453.484,Z 383.998,A -85,B 0,C 180,E1 -8494.779,E2 -8494.779} C_VEL
LIN {X 0,Y 453.481,Z 384,A -85,B 0,C 180,E1 -8498.31,E2 -8498.31} C_VEL
LIN {X 0,Y 453.511,Z 383.995,A -85,B 0,C 180,E1 -8500.607,E2 -8500.607} C_VEL
LIN {X 0,Y 453.462,Z 384.002,A -85,B 0,C 180,E1 -8504.222,E2 -8504.222} C_VEL
LIN {X 0,Y 453.46,Z 384,A -85,B 0,C 180,E1 -8507.006,E2 -8507.006} C_VEL
LIN {X 0,Y 453.515,Z 383.994,A -85,B 0,C 180,E1 -8510.554,E2 -8510.554} C_VEL
LIN {X 0,Y 453.455,Z 384.003,A -85,B 0,C 180,E1 -8513.918,E2 -8513.918} C_VEL
LIN {X 0,Y 453.482,Z 383.997,A -85,B 0,C 180,E1 -8517.152,E2 -8517.152} C_VEL
LIN {X 0,Y 453.475,Z 384.001,A -85,B 0,C 180,E1 -8520.269,E2 -8520.269} C_VEL
LIN {X 0,Y 453.507,Z 383.994,A -85,B 0,C 180,E1 -8523.295,E2 -8523.295} C_VEL
LIN {X 0,Y 453.505,Z 383.996,A -85,B 0,C 180,E1 -8526.24,E2 -8526.24} C_VEL
LIN {X 0,Y 453.485,Z 383.997,A -85,B 0,C 180,E1 -8529.118,E2 -8529.118} C_VEL
LIN {X 0,Y 453.513,Z 383.996,A -85,B 0,C 180,E1 -8531.945,E2 -8531.945} C_VEL
LIN {X 0,Y 453.543,Z 383.99,A -85,B 0,C 180,E1 -8534.727,E2 -8534.727} C_VEL
LIN {X 0,Y 453.563,Z 383.988,A -85,B 0,C 180,E1 -8538.38,E2 -8538.38} C_VEL
LIN {X 0,Y 453.656,Z 383.978,A -85,B 0,C 180,E1 -8541.986,E2 -8541.986} C_VEL
LIN {X 0,Y 453.641,Z 383.976,A -85,B 0,C 180,E1 -8543.094,E2 -8543.094} C_VEL
LIN {X 0,Y 452.95,Z 384.066,A -85,B 0,C 180,E1 -8543.834,E2 -8543.834} C_VEL
LIN {X 0,Y 449.968,Z 384.436,A -85,B 0,C 180,E1 -8545.035,E2 -8545.035} C_VEL
LIN {X 0,Y 447.492,Z 384.745,A -85,B 0,C 180,E1 -8546.004,E2 -8546.004} C_VEL
LIN {X 0,Y 446.501,Z 384.867,A -85,B 0,C 180,E1 -8546.755,E2 -8546.755} C_VEL
LIN {X 0,Y 446.46,Z 384.872,A -85,B 0,C 180,E1 -8547.008,E2 -8547.008} C_VEL
LIN {X 0,Y 446.505,Z 384.87,A -85,B 0,C 180,E1 -8549.098,E2 -8549.098} C_VEL
LIN {X 0,Y 446.002,Z 385.094,A -85,B 0,C 180,E1 -8550.903,E2 -8550.903} C_VEL
LIN {X 0,Y 445.977,Z 388.79,A -85,B 0,C 180,E1 -8554.519,E2 -8554.519} C_VEL
LIN {X 0,Y 445.904,Z 391.595,A -85,B 0,C 180,E1 -8557.244,E2 -8557.244} C_VEL
LIN {X 0,Y 445.775,Z 395.504,A -85,B 0,C 180,E1 -8560.905,E2 -8560.905} C_VEL
LIN {X 0,Y 445.675,Z 398.424,A -85,B 0,C 180,E1 -8563.682,E2 -8563.682} C_VEL
LIN {X 0,Y 445.631,Z 400.926,A -85,B 0,C 180,E1 -8565.983,E2 -8565.983} C_VEL
LIN {X 0,Y 448.832,Z 414.31,A -85,B 0,C 180,E1 -8566.528,E2 -8566.528} C_VEL
LIN {X 0,Y 449.721,Z 418.364,A -85,B 0,C 180,E1 -8566.73,E2 -8566.73} C_VEL
LIN {X 0,Y 449.237,Z 431.256,A -85,B 0,C 180,E1 -8567.387,E2 -8567.387} C_VEL
LIN {X 0,Y 448.759,Z 442.19,A -85,B 0,C 180,E1 -8568.123,E2 -8568.123} C_VEL
LIN {X 0,Y 448.208,Z 453.596,A -85,B 0,C 180,E1 -8569.106,E2 -8569.106} C_VEL
LIN {X 0,Y 447.583,Z 463.877,A -85,B 0,C 180,E1 -8570.209,E2 -8570.209} C_VEL
LIN {X 0,Y 447.03,Z 472.828,A -85,B 0,C 180,E1 -8571.396,E2 -8571.396} C_VEL
LIN {X 0,Y 446.587,Z 480.652,A -85,B 0,C 180,E1 -8572.678,E2 -8572.678} C_VEL
LIN {X 0,Y 446.155,Z 487.987,A -85,B 0,C 180,E1 -8574.177,E2 -8574.177} C_VEL
LIN {X 0,Y 445.87,Z 493.489,A -85,B 0,C 180,E1 -8575.609,E2 -8575.609} C_VEL
LIN {X 0,Y 445.719,Z 498.103,A -85,B 0,C 180,E1 -8577.21,E2 -8577.21} C_VEL
LIN {X 0,Y 445.555,Z 500.336,A -85,B 0,C 180,E1 -8578.242,E2 -8578.242} C_VEL
LIN {X 0,Y 445.412,Z 502.667,A -85,B 0,C 180,E1 -8579.792,E2 -8579.792} C_VEL
LIN {X 0,Y 445.366,Z 503.845,A -85,B 0,C 180,E1 -8581.555,E2 -8581.555} C_VEL
LIN {X 0,Y 445.391,Z 503.587,A -85,B 0,C 180,E1 -8583.247,E2 -8583.247} C_VEL
LIN {X 0,Y 445.49,Z 502.044,A -85,B 0,C 180,E1 -8584.88,E2 -8584.88} C_VEL
LIN {X 0,Y 445.622,Z 499.279,A -85,B 0,C 180,E1 -8586.454,E2 -8586.454} C_VEL
LIN {X 0,Y 445.842,Z 495.302,A -85,B 0,C 180,E1 -8587.985,E2 -8587.985} C_VEL
LIN {X 0,Y 446.142,Z 490.099,A -85,B 0,C 180,E1 -8589.476,E2 -8589.476} C_VEL
LIN {X 0,Y 446.504,Z 483.6,A -85,B 0,C 180,E1 -8590.929,E2 -8590.929} C_VEL
LIN {X 0,Y 446.956,Z 475.521,A -85,B 0,C 180,E1 -8592.35,E2 -8592.35} C_VEL
LIN {X 0,Y 447.56,Z 465.877,A -85,B 0,C 180,E1 -8593.703,E2 -8593.703} C_VEL
LIN {X 0,Y 448.07,Z 456.763,A -85,B 0,C 180,E1 -8594.737,E2 -8594.737} C_VEL
LIN {X 0,Y 448.613,Z 446.385,A -85,B 0,C 180,E1 -8595.69,E2 -8595.69} C_VEL
LIN {X 0,Y 449.183,Z 434.228,A -85,B 0,C 180,E1 -8596.572,E2 -8596.572} C_VEL
LIN {X 0,Y 449.648,Z 423.117,A -85,B 0,C 180,E1 -8597.191,E2 -8597.191} C_VEL
LIN {X 0,Y 449.776,Z 419.326,A -85,B 0,C 180,E1 -8597.363,E2 -8597.363} C_VEL
LIN {X 0,Y 447.327,Z 408.319,A -85,B 0,C 180,E1 -8597.88,E2 -8597.88} C_VEL
LIN {X 0,Y 445.628,Z 401.688,A -85,B 0,C 180,E1 -8598.138,E2 -8598.138} C_VEL
LIN {X 0,Y 445.648,Z 398.856,A -85,B 0,C 180,E1 -8600.89,E2 -8600.89} C_VEL
LIN {X 0,Y 445.772,Z 395.369,A -85,B 0,C 180,E1 -8604.314,E2 -8604.314} C_VEL
LIN {X 0,Y 445.879,Z 392.045,A -85,B 0,C 180,E1 -8607.594,E2 -8607.594} C_VEL
LIN {X 0,Y 445.955,Z 388.904,A -85,B 0,C 180,E1 -8610.755,E2 -8610.755} C_VEL
LIN {X 0,Y 446.04,Z 385.774,A -85,B 0,C 180,E1 -8613.91,E2 -8613.91} C_VEL
LIN {X 0,Y 446.078,Z 384.926,A -85,B 0,C 180,E1 -8614.825,E2 -8614.825} C_VEL
LIN {X 0,Y 446.378,Z 384.887,A -85,B 0,C 180,E1 -8617.798,E2 -8617.798} C_VEL
LIN {X 0,Y 446.47,Z 384.874,A -85,B 0,C 180,E1 -8620.814,E2 -8620.814} C_VEL
LIN {X 0,Y 446.491,Z 384.869,A -85,B 0,C 180,E1 -8623.772,E2 -8623.772} C_VEL
LIN {X 0,Y 446.51,Z 384.868,A -85,B 0,C 180,E1 -8627.384,E2 -8627.384} C_VEL
LIN {X 0,Y 446.533,Z 384.865,A -85,B 0,C 180,E1 -8630.944,E2 -8630.944} C_VEL
LIN {X 0,Y 446.641,Z 384.851,A -85,B 0,C 180,E1 -8633.676,E2 -8633.676} C_VEL
LIN {X 0,Y 446.703,Z 384.84,A -85,B 0,C 180,E1 -8637.295,E2 -8637.295} C_VEL
LIN {X 0,Y 446.787,Z 384.831,A -85,B 0,C 180,E1 -8640,E2 -8640} C_VEL
LIN {X 0,Y 446.703,Z 384.842,A -85,B 0,C 180,E1 -8642.705,E2 -8642.705} C_VEL
LIN {X 0,Y 446.64,Z 384.852,A -85,B 0,C 180,E1 -8646.324,E2 -8646.324} C_VEL
LIN {X 0,Y 446.533,Z 384.865,A -85,B 0,C 180,E1 -8649.055,E2 -8649.055} C_VEL
LIN {X 0,Y 446.515,Z 384.865,A -85,B 0,C 180,E1 -8652.73,E2 -8652.73} C_VEL
LIN {X 0,Y 446.491,Z 384.868,A -85,B 0,C 180,E1 -8656.228,E2 -8656.228} C_VEL
LIN {X 0,Y 446.464,Z 384.87,A -85,B 0,C 180,E1 -8659.303,E2 -8659.303} C_VEL
LIN {X 0,Y 446.413,Z 384.881,A -85,B 0,C 180,E1 -8662.2,E2 -8662.2} C_VEL
LIN {X 0,Y 446.453,Z 384.874,A -85,B 0,C 180,E1 -8665.153,E2 -8665.153} C_VEL
LIN {X 0,Y 446.48,Z 384.872,A -85,B 0,C 180,E1 -8668.179,E2 -8668.179} C_VEL
LIN {X 0,Y 446.414,Z 384.882,A -85,B 0,C 180,E1 -8671.775,E2 -8671.775} C_VEL
LIN {X 0,Y 446.418,Z 384.881,A -85,B 0,C 180,E1 -8674.524,E2 -8674.524} C_VEL
LIN {X 0,Y 446.435,Z 384.879,A -85,B 0,C 180,E1 -8678.083,E2 -8678.083} C_VEL
LIN {X 0,Y 446.441,Z 384.877,A -85,B 0,C 180,E1 -8680.921,E2 -8680.921} C_VEL
LIN {X 0,Y 446.399,Z 384.883,A -85,B 0,C 180,E1 -8683.846,E2 -8683.846} C_VEL
LIN {X 0,Y 446.397,Z 384.885,A -85,B 0,C 180,E1 -8686.404,E2 -8686.404} C_VEL
LIN {X 0,Y 446.469,Z 385.011,A -85,B 0,C 180,E1 -8688.162,E2 -8688.162} C_VEL
LIN {X 0,Y 447.493,Z 390.762,A -85,B 0,C 180,E1 -8691.082,E2 -8691.082} C_VEL
LIN {X 0,Y 448.37,Z 395.759,A -85,B 0,C 180,E1 -8693.443,E2 -8693.443} C_VEL
LIN {X 0,Y 448.229,Z 400.843,A -85,B 0,C 180,E1 -8695.636,E2 -8695.636} C_VEL
LIN {X 0,Y 447.738,Z 407.527,A -85,B 0,C 180,E1 -8698.368,E2 -8698.368} C_VEL
LIN {X 0,Y 447.254,Z 416.478,A -85,B 0,C 180,E1 -8701.874,E2 -8701.874} C_VEL
LIN {X 0,Y 446.838,Z 424.441,A -85,B 0,C 180,E1 -8704.871,E2 -8704.871} C_VEL
LIN {X 0,Y 446.486,Z 433.758,A -85,B 0,C 180,E1 -8708.234,E2 -8708.234} C_VEL
LIN {X 0,Y 446.253,Z 442.39,A -85,B 0,C 180,E1 -8711.264,E2 -8711.264} C_VEL
LIN {X 0,Y 446.006,Z 449.719,A -85,B 0,C 180,E1 -8713.819,E2 -8713.819} C_VEL
LIN {X 0,Y 448.298,Z 463.989,A -85,B 0,C 180,E1 -8714.307,E2 -8714.307} C_VEL
LIN {X 0,Y 449.41,Z 472.739,A -85,B 0,C 180,E1 -8714.699,E2 -8714.699} C_VEL
LIN {X 0,Y 448.95,Z 483.801,A -85,B 0,C 180,E1 -8715.263,E2 -8715.263} C_VEL
LIN {X 0,Y 448.332,Z 495.709,A -85,B 0,C 180,E1 -8716.054,E2 -8716.054} C_VEL
LIN {X 0,Y 447.79,Z 506.779,A -85,B 0,C 180,E1 -8716.998,E2 -8716.998} C_VEL
LIN {X 0,Y 447.309,Z 516.171,A -85,B 0,C 180,E1 -8717.984,E2 -8717.984} C_VEL
LIN {X 0,Y 446.689,Z 525.076,A -85,B 0,C 180,E1 -8719.117,E2 -8719.117} C_VEL
LIN {X 0,Y 446.24,Z 533.778,A -85,B 0,C 180,E1 -8720.481,E2 -8720.481} C_VEL
LIN {X 0,Y 445.884,Z 540.735,A -85,B 0,C 180,E1 -8721.845,E2 -8721.845} C_VEL
LIN {X 0,Y 445.649,Z 546.318,A -85,B 0,C 180,E1 -8723.208,E2 -8723.208} C_VEL
LIN {X 0,Y 445.541,Z 550.699,A -85,B 0,C 180,E1 -8724.569,E2 -8724.569} C_VEL
LIN {X 0,Y 445.427,Z 553.016,A -85,B 0,C 180,E1 -8725.475,E2 -8725.475} C_VEL
LIN {X 0,Y 445.398,Z 554.9,A -85,B 0,C 180,E1 -8726.381,E2 -8726.381} C_VEL
LIN {X 0,Y 445.423,Z 556.315,A -85,B 0,C 180,E1 -8727.287,E2 -8727.287} C_VEL
LIN {X 0,Y 445.372,Z 557.938,A -85,B 0,C 180,E1 -8729.096,E2 -8729.096} C_VEL
LIN {X 0,Y 445.349,Z 558.159,A -85,B 0,C 180,E1 -8730,E2 -8730} C_VEL
LIN {X 0,Y 445.372,Z 557.944,A -85,B 0,C 180,E1 -8730.904,E2 -8730.904} C_VEL
LIN {X 0,Y 445.422,Z 556.333,A -85,B 0,C 180,E1 -8732.713,E2 -8732.713} C_VEL
LIN {X 0,Y 445.397,Z 554.924,A -85,B 0,C 180,E1 -8733.618,E2 -8733.618} C_VEL
LIN {X 0,Y 445.5,Z 551.969,A -85,B 0,C 180,E1 -8734.977,E2 -8734.977} C_VEL
LIN {X 0,Y 445.584,Z 547.597,A -85,B 0,C 180,E1 -8736.448,E2 -8736.448} C_VEL
LIN {X 0,Y 445.804,Z 541.81,A -85,B 0,C 180,E1 -8737.928,E2 -8737.928} C_VEL
LIN {X 0,Y 446.185,Z 535.095,A -85,B 0,C 180,E1 -8739.291,E2 -8739.291} C_VEL
LIN {X 0,Y 446.606,Z 526.766,A -85,B 0,C 180,E1 -8740.655,E2 -8740.655} C_VEL
LIN {X 0,Y 447.174,Z 518.239,A -85,B 0,C 180,E1 -8741.789,E2 -8741.789} C_VEL
LIN {X 0,Y 447.724,Z 508.414,A -85,B 0,C 180,E1 -8742.856,E2 -8742.856} C_VEL
LIN {X 0,Y 448.259,Z 497.29,A -85,B 0,C 180,E1 -8743.833,E2 -8743.833} C_VEL
LIN {X 0,Y 448.836,Z 485.893,A -85,B 0,C 180,E1 -8744.624,E2 -8744.624} C_VEL
LIN {X 0,Y 449.4,Z 474.21,A -85,B 0,C 180,E1 -8745.243,E2 -8745.243} C_VEL
LIN {X 0,Y 448.899,Z 467.916,A -85,B 0,C 180,E1 -8745.53,E2 -8745.53} C_VEL
LIN {X 0,Y 446.701,Z 454.409,A -85,B 0,C 180,E1 -8746.038,E2 -8746.038} C_VEL
LIN {X 0,Y 446.006,Z 449.989,A -85,B 0,C 180,E1 -8746.181,E2 -8746.181} C_VEL
LIN {X 0,Y 446.329,Z 441.156,A -85,B 0,C 180,E1 -8749.309,E2 -8749.309} C_VEL
LIN {X 0,Y 446.57,Z 433.034,A -85,B 0,C 180,E1 -8752.191,E2 -8752.191} C_VEL
LIN {X 0,Y 446.907,Z 424.932,A -85,B 0,C 180,E1 -8755.124,E2 -8755.124} C_VEL
LIN {X 0,Y 447.359,Z 416.296,A -85,B 0,C 180,E1 -8758.386,E2 -8758.386} C_VEL
LIN {X 0,Y 447.886,Z 406.874,A -85,B 0,C 180,E1 -8762.076,E2 -8762.076} C_VEL
LIN {X 0,Y 448.327,Z 400.005,A -85,B 0,C 180,E1 -8764.89,E2 -8764.89} C_VEL
LIN {X 0,Y 448.436,Z 396.097,A -85,B 0,C 180,E1 -8766.55,E2 -8766.55} C_VEL
LIN {X 0,Y 447.281,Z 389.347,A -85,B 0,C 180,E1 -8769.653,E2 -8769.653} C_VEL
LIN {X 0,Y 446.44,Z 384.876,A -85,B 0,C 180,E1 -8771.841,E2 -8771.841} C_VEL
LIN {X 0,Y 446.449,Z 384.877,A -85,B 0,C 180,E1 -8775.103,E2 -8775.103} C_VEL
LIN {X 0,Y 446.43,Z 384.878,A -85,B 0,C 180,E1 -8778.609,E2 -8778.609} C_VEL
LIN {X 0,Y 446.469,Z 384.873,A -85,B 0,C 180,E1 -8780.975,E2 -8780.975} C_VEL
LIN {X 0,Y 446.415,Z 384.879,A -85,B 0,C 180,E1 -8784.373,E2 -8784.373} C_VEL
LIN {X 0,Y 446.416,Z 384.877,A -85,B 0,C 180,E1 -8787.638,E2 -8787.638} C_VEL
LIN {X 0,Y 446.442,Z 384.877,A -85,B 0,C 180,E1 -8790.79,E2 -8790.79} C_VEL
LIN {X 0,Y 446.47,Z 384.871,A -85,B 0,C 180,E1 -8793.848,E2 -8793.848} C_VEL
LIN {X 0,Y 446.421,Z 384.879,A -85,B 0,C 180,E1 -8796.823,E2 -8796.823} C_VEL
LIN {X 0,Y 446.436,Z 384.874,A -85,B 0,C 180,E1 -8799.737,E2 -8799.737} C_VEL
LIN {X 0,Y 446.455,Z 384.875,A -85,B 0,C 180,E1 -8802.597,E2 -8802.597} C_VEL
LIN {X 0,Y 446.461,Z 384.872,A -85,B 0,C 180,E1 -8805.412,E2 -8805.412} C_VEL
LIN {X 0,Y 446.51,Z 384.866,A -85,B 0,C 180,E1 -8808.193,E2 -8808.193} C_VEL
LIN {X 0,Y 446.591,Z 384.856,A -85,B 0,C 180,E1 -8811.858,E2 -8811.858} C_VEL
LIN {X 0,Y 446.636,Z 384.852,A -85,B 0,C 180,E1 -8814.583,E2 -8814.583} C_VEL
LIN {X 0,Y 446.7,Z 384.842,A -85,B 0,C 180,E1 -8817.295,E2 -8817.295} C_VEL
LIN {X 0,Y 446.785,Z 384.832,A -85,B 0,C 180,E1 -8820,E2 -8820} C_VEL
LIN {X 0,Y 446.701,Z 384.845,A -85,B 0,C 180,E1 -8822.705,E2 -8822.705} C_VEL
LIN {X 0,Y 446.637,Z 384.853,A -85,B 0,C 180,E1 -8826.324,E2 -8826.324} C_VEL
LIN {X 0,Y 446.53,Z 384.865,A -85,B 0,C 180,E1 -8829.056,E2 -8829.056} C_VEL
LIN {X 0,Y 446.512,Z 384.868,A -85,B 0,C 180,E1 -8832.73,E2 -8832.73} C_VEL
LIN {X 0,Y 446.488,Z 384.872,A -85,B 0,C 180,E1 -8836.228,E2 -8836.228} C_VEL
LIN {X 0,Y 446.461,Z 384.872,A -85,B 0,C 180,E1 -8839.304,E2 -8839.304} C_VEL
LIN {X 0,Y 446.411,Z 384.88,A -85,B 0,C 180,E1 -8842.2,E2 -8842.2} C_VEL
LIN {X 0,Y 446.451,Z 384.872,A -85,B 0,C 180,E1 -8845.153,E2 -8845.153} C_VEL
LIN {X 0,Y 446.478,Z 384.873,A -85,B 0,C 180,E1 -8848.179,E2 -8848.179} C_VEL
LIN {X 0,Y 446.413,Z 384.879,A -85,B 0,C 180,E1 -8851.776,E2 -8851.776} C_VEL
LIN {X 0,Y 446.425,Z 384.879,A -85,B 0,C 180,E1 -8854.524,E2 -8854.524} C_VEL
LIN {X 0,Y 446.434,Z 384.878,A -85,B 0,C 180,E1 -8858.084,E2 -8858.084} C_VEL
LIN {X 0,Y 446.439,Z 384.875,A -85,B 0,C 180,E1 -8860.921,E2 -8860.921} C_VEL
LIN {X 0,Y 446.397,Z 384.882,A -85,B 0,C 180,E1 -8863.847,E2 -8863.847} C_VEL
LIN {X 0,Y 446.396,Z 384.882,A -85,B 0,C 180,E1 -8866.404,E2 -8866.404} C_VEL
LIN {X 0,Y 446.424,Z 384.876,A -85,B 0,C 180,E1 -8869.083,E2 -8869.083} C_VEL
LIN {X 0,Y 446.428,Z 384.878,A -85,B 0,C 180,E1 -8871.919,E2 -8871.919} C_VEL
LIN {X 0,Y 446.429,Z 384.876,A -85,B 0,C 180,E1 -8875.478,E2 -8875.478} C_VEL
LIN {X 0,Y 446.416,Z 384.878,A -85,B 0,C 180,E1 -8878.701,E2 -8878.701} C_VEL
LIN {X 0,Y 446.485,Z 384.871,A -85,B 0,C 180,E1 -8881.822,E2 -8881.822} C_VEL
LIN {X 0,Y 446.459,Z 384.872,A -85,B 0,C 180,E1 -8884.849,E2 -8884.849} C_VEL
LIN {X 0,Y 446.45,Z 384.875,A -85,B 0,C 180,E1 -8888.246,E2 -8888.246} C_VEL
LIN {X 0,Y 446.459,Z 384.875,A -85,B 0,C 180,E1 -8891.65,E2 -8891.65} C_VEL
LIN {X 0,Y 446.511,Z 384.867,A -85,B 0,C 180,E1 -8894.48,E2 -8894.48} C_VEL
LIN {X 0,Y 446.521,Z 384.866,A -85,B 0,C 180,E1 -8898.194,E2 -8898.194} C_VEL
LIN {X 0,Y 446.604,Z 384.856,A -85,B 0,C 180,E1 -8901.858,E2 -8901.858} C_VEL
LIN {X 0,Y 446.649,Z 384.848,A -85,B 0,C 180,E1 -8904.583,E2 -8904.583} C_VEL
LIN {X 0,Y 446.46,Z 384.872,A -85,B 0,C 180,E1 -8907.008,E2 -8907.008} C_VEL
LIN {X 0,Y 446.211,Z 384.923,A -85,B 0,C 180,E1 -8907.513,E2 -8907.513} C_VEL
LIN {X 0,Y 444.863,Z 385.129,A -85,B 0,C 180,E1 -8908.257,E2 -8908.257} C_VEL
LIN {X 0,Y 440.267,Z 385.647,A -85,B 0,C 180,E1 -8909.97,E2 -8909.97} C_VEL
LIN {X 0,Y 438.97,Z 385.869,A -85,B 0,C 180,E1 -8910.86,E2 -8910.86} C_VEL
LIN {X 0,Y 438.923,Z 385.97,A -85,B 0,C 180,E1 -8910.988,E2 -8910.988} C_VEL
LIN {X 0,Y 438.918,Z 389.603,A -85,B 0,C 180,E1 -8914.592,E2 -8914.592} C_VEL
LIN {X 0,Y 438.836,Z 392.464,A -85,B 0,C 180,E1 -8917.361,E2 -8917.361} C_VEL
LIN {X 0,Y 438.707,Z 396.376,A -85,B 0,C 180,E1 -8921.083,E2 -8921.083} C_VEL
LIN {X 0,Y 438.593,Z 399.399,A -85,B 0,C 180,E1 -8923.908,E2 -8923.908} C_VEL
LIN {X 0,Y 438.592,Z 401.301,A -85,B 0,C 180,E1 -8925.718,E2 -8925.718} C_VEL
LIN {X 0,Y 442.052,Z 415.762,A -85,B 0,C 180,E1 -8926.33,E2 -8926.33} C_VEL
LIN {X 0,Y 442.851,Z 419.872,A -85,B 0,C 180,E1 -8926.542,E2 -8926.542} C_VEL
LIN {X 0,Y 442.373,Z 432.275,A -85,B 0,C 180,E1 -8927.196,E2 -8927.196} C_VEL
LIN {X 0,Y 441.865,Z 443.109,A -85,B 0,C 180,E1 -8927.949,E2 -8927.949} C_VEL
LIN {X 0,Y 441.289,Z 454.299,A -85,B 0,C 180,E1 -8928.935,E2 -8928.935} C_VEL
LIN {X 0,Y 440.679,Z 463.834,A -85,B 0,C 180,E1 -8929.971,E2 -8929.971} C_VEL
LIN {X 0,Y 440.155,Z 472.027,A -85,B 0,C 180,E1 -8931.055,E2 -8931.055} C_VEL
LIN {X 0,Y 439.686,Z 479.515,A -85,B 0,C 180,E1 -8932.25,E2 -8932.25} C_VEL
LIN {X 0,Y 439.258,Z 486.319,A -85,B 0,C 180,E1 -8933.577,E2 -8933.577} C_VEL
LIN {X 0,Y 438.906,Z 492.51,A -85,B 0,C 180,E1 -8935.108,E2 -8935.108} C_VEL
LIN {X 0,Y 438.701,Z 497.293,A -85,B 0,C 180,E1 -8936.651,E2 -8936.651} C_VEL
LIN {X 0,Y 438.481,Z 500.736,A -85,B 0,C 180,E1 -8938.17,E2 -8938.17} C_VEL
LIN {X 0,Y 438.326,Z 503.354,A -85,B 0,C 180,E1 -8940.023,E2 -8940.023} C_VEL
LIN {X 0,Y 438.281,Z 504.327,A -85,B 0,C 180,E1 -8941.801,E2 -8941.801} C_VEL
LIN {X 0,Y 438.319,Z 503.899,A -85,B 0,C 180,E1 -8943.512,E2 -8943.512} C_VEL
LIN {X 0,Y 438.439,Z 502.018,A -85,B 0,C 180,E1 -8945.244,E2 -8945.244} C_VEL
LIN {X 0,Y 438.582,Z 499.207,A -85,B 0,C 180,E1 -8946.753,E2 -8946.753} C_VEL
LIN {X 0,Y 438.823,Z 495.08,A -85,B 0,C 180,E1 -8948.301,E2 -8948.301} C_VEL
LIN {X 0,Y 439.149,Z 489.724,A -85,B 0,C 180,E1 -8949.809,E2 -8949.809} C_VEL
LIN {X 0,Y 439.559,Z 482.979,A -85,B 0,C 180,E1 -8951.281,E2 -8951.281} C_VEL
LIN {X 0,Y 440.087,Z 474.633,A -85,B 0,C 180,E1 -8952.726,E2 -8952.726} C_VEL
LIN {X 0,Y 440.667,Z 466.137,A -85,B 0,C 180,E1 -8953.915,E2 -8953.915} C_VEL
LIN {X 0,Y 441.198,Z 456.839,A -85,B 0,C 180,E1 -8954.98,E2 -8954.98} C_VEL
LIN {X 0,Y 441.825,Z 445.288,A -85,B 0,C 180,E1 -8956.035,E2 -8956.035} C_VEL
LIN {X 0,Y 442.361,Z 434.286,A -85,B 0,C 180,E1 -8956.831,E2 -8956.831} C_VEL
LIN {X 0,Y 442.879,Z 422.946,A -85,B 0,C 180,E1 -8957.464,E2 -8957.464} C_VEL
LIN {X 0,Y 442.761,Z 419.027,A -85,B 0,C 180,E1 -8957.651,E2 -8957.651} C_VEL
LIN {X 0,Y 439.65,Z 406.32,A -85,B 0,C 180,E1 -8958.249,E2 -8958.249} C_VEL
LIN {X 0,Y 438.575,Z 402.135,A -85,B 0,C 180,E1 -8958.415,E2 -8958.415} C_VEL
LIN {X 0,Y 438.598,Z 398.752,A -85,B 0,C 180,E1 -8961.735,E2 -8961.735} C_VEL
LIN {X 0,Y 438.726,Z 395.671,A -85,B 0,C 180,E1 -8964.782,E2 -8964.782} C_VEL
LIN {X 0,Y 438.857,Z 392.39,A -85,B 0,C 180,E1 -8968.097,E2 -8968.097} C_VEL
LIN {X 0,Y 438.924,Z 389.215,A -85,B 0,C 180,E1 -8971.291,E2 -8971.291} C_VEL
LIN {X 0,Y 438.998,Z 386.194,A -85,B 0,C 180,E1 -8974.389,E2 -8974.389} C_VEL
LIN {X 0,Y 439.216,Z 385.78,A -85,B 0,C 180,E1 -8976.42,E2 -8976.42} C_VEL
LIN {X 0,Y 439.406,Z 385.757,A -85,B 0,C 180,E1 -8978.416,E2 -8978.416} C_VEL
LIN {X 0,Y 439.423,Z 385.75,A -85,B 0,C 180,E1 -8981.345,E2 -8981.345} C_VEL
LIN {X 0,Y 439.457,Z 385.746,A -85,B 0,C 180,E1 -8984.224,E2 -8984.224} C_VEL
LIN {X 0,Y 439.479,Z 385.744,A -85,B 0,C 180,E1 -8988.001,E2 -8988.001} C_VEL
LIN {X 0,Y 439.542,Z 385.737,A -85,B 0,C 180,E1 -8991.726,E2 -8991.726} C_VEL
LIN {X 0,Y 439.615,Z 385.725,A -85,B 0,C 180,E1 -8994.496,E2 -8994.496} C_VEL
LIN {X 0,Y 439.629,Z 385.725,A -85,B 0,C 180,E1 -8998.168,E2 -8998.168} C_VEL
LIN {X 0,Y 439.757,Z 385.706,A -85,B 0,C 180,E1 -9000,E2 -9000} C_VEL
LIN {X 0,Y 439.65,Z 385.721,A -85,B 0,C 180,E1 -9002.749,E2 -9002.749} C_VEL
LIN {X 0,Y 439.611,Z 385.729,A -85,B 0,C 180,E1 -9006.425,E2 -9006.425} C_VEL
LIN {X 0,Y 439.495,Z 385.741,A -85,B 0,C 180,E1 -9009.202,E2 -9009.202} C_VEL
LIN {X 0,Y 439.46,Z 385.743,A -85,B 0,C 180,E1 -9012.938,E2 -9012.938} C_VEL
LIN {X 0,Y 439.442,Z 385.746,A -85,B 0,C 180,E1 -9016.349,E2 -9016.349} C_VEL
LIN {X 0,Y 439.397,Z 385.753,A -85,B 0,C 180,E1 -9019.627,E2 -9019.627} C_VEL
LIN {X 0,Y 439.36,Z 385.758,A -85,B 0,C 180,E1 -9022.576,E2 -9022.576} C_VEL
LIN {X 0,Y 439.401,Z 385.754,A -85,B 0,C 180,E1 -9025.585,E2 -9025.585} C_VEL
LIN {X 0,Y 439.413,Z 385.749,A -85,B 0,C 180,E1 -9028.674,E2 -9028.674} C_VEL
LIN {X 0,Y 439.364,Z 385.76,A -85,B 0,C 180,E1 -9032.03,E2 -9032.03} C_VEL
LIN {X 0,Y 439.388,Z 385.757,A -85,B 0,C 180,E1 -9035.34,E2 -9035.34} C_VEL
LIN {X 0,Y 439.395,Z 385.755,A -85,B 0,C 180,E1 -9038.594,E2 -9038.594} C_VEL
LIN {X 0,Y 439.396,Z 385.756,A -85,B 0,C 180,E1 -9041.259,E2 -9041.259} C_VEL
LIN {X 0,Y 439.399,Z 385.754,A -85,B 0,C 180,E1 -9044.73,E2 -9044.73} C_VEL
LIN {X 0,Y 439.423,Z 385.884,A -85,B 0,C 180,E1 -9047.8,E2 -9047.8} C_VEL
LIN {X 0,Y 440.305,Z 390.691,A -85,B 0,C 180,E1 -9050.323,E2 -9050.323} C_VEL
LIN {X 0,Y 441.397,Z 396.969,A -85,B 0,C 180,E1 -9053.361,E2 -9053.361} C_VEL
LIN {X 0,Y 441.241,Z 401.828,A -85,B 0,C 180,E1 -9055.526,E2 -9055.526} C_VEL
LIN {X 0,Y 440.731,Z 408.359,A -85,B 0,C 180,E1 -9058.25,E2 -9058.25} C_VEL
LIN {X 0,Y 440.303,Z 416.206,A -85,B 0,C 180,E1 -9061.39,E2 -9061.39} C_VEL
LIN {X 0,Y 439.836,Z 424.129,A -85,B 0,C 180,E1 -9064.442,E2 -9064.442} C_VEL
LIN {X 0,Y 439.504,Z 432.159,A -85,B 0,C 180,E1 -9067.432,E2 -9067.432} C_VEL
LIN {X 0,Y 439.224,Z 441.33,A -85,B 0,C 180,E1 -9070.745,E2 -9070.745} C_VEL
LIN {X 0,Y 438.927,Z 449.283,A -85,B 0,C 180,E1 -9073.563,E2 -9073.563} C_VEL
LIN {X 0,Y 441.062,Z 462.856,A -85,B 0,C 180,E1 -9074.02,E2 -9074.02} C_VEL
LIN {X 0,Y 442.492,Z 473.565,A -85,B 0,C 180,E1 -9074.513,E2 -9074.513} C_VEL
LIN {X 0,Y 441.96,Z 485.263,A -85,B 0,C 180,E1 -9075.142,E2 -9075.142} C_VEL
LIN {X 0,Y 441.323,Z 496.675,A -85,B 0,C 180,E1 -9075.945,E2 -9075.945} C_VEL
LIN {X 0,Y 440.789,Z 506.831,A -85,B 0,C 180,E1 -9076.84,E2 -9076.84} C_VEL
LIN {X 0,Y 440.326,Z 515.708,A -85,B 0,C 180,E1 -9077.791,E2 -9077.791} C_VEL
LIN {X 0,Y 439.679,Z 524.616,A -85,B 0,C 180,E1 -9078.941,E2 -9078.941} C_VEL
LIN {X 0,Y 439.186,Z 533.323,A -85,B 0,C 180,E1 -9080.327,E2 -9080.327} C_VEL
LIN {X 0,Y 438.82,Z 540.285,A -85,B 0,C 180,E1 -9081.712,E2 -9081.712} C_VEL
LIN {X 0,Y 438.566,Z 545.871,A -85,B 0,C 180,E1 -9083.097,E2 -9083.097} C_VEL
LIN {X 0,Y 438.461,Z 550.258,A -85,B 0,C 180,E1 -9084.481,E2 -9084.481} C_VEL
LIN {X 0,Y 438.357,Z 552.579,A -85,B 0,C 180,E1 -9085.402,E2 -9085.402} C_VEL
LIN {X 0,Y 438.304,Z 554.463,A -85,B 0,C 180,E1 -9086.322,E2 -9086.322} C_VEL
LIN {X 0,Y 438.351,Z 555.882,A -85,B 0,C 180,E1 -9087.243,E2 -9087.243} C_VEL
LIN {X 0,Y 438.283,Z 557.508,A -85,B 0,C 180,E1 -9089.081,E2 -9089.081} C_VEL
LIN {X 0,Y 438.29,Z 557.731,A -85,B 0,C 180,E1 -9090,E2 -9090} C_VEL
LIN {X 0,Y 438.283,Z 557.516,A -85,B 0,C 180,E1 -9090.919,E2 -9090.919} C_VEL
LIN {X 0,Y 438.351,Z 555.907,A -85,B 0,C 180,E1 -9092.757,E2 -9092.757} C_VEL
LIN {X 0,Y 438.302,Z 554.498,A -85,B 0,C 180,E1 -9093.677,E2 -9093.677} C_VEL
LIN {X 0,Y 438.434,Z 551.544,A -85,B 0,C 180,E1 -9095.058,E2 -9095.058} C_VEL
LIN {X 0,Y 438.505,Z 547.539,A -85,B 0,C 180,E1 -9096.441,E2 -9096.441} C_VEL
LIN {X 0,Y 438.753,Z 541.384,A -85,B 0,C 180,E1 -9098.057,E2 -9098.057} C_VEL
LIN {X 0,Y 439.152,Z 534.668,A -85,B 0,C 180,E1 -9099.441,E2 -9099.441} C_VEL
LIN {X 0,Y 439.59,Z 526.338,A -85,B 0,C 180,E1 -9100.827,E2 -9100.827} C_VEL
LIN {X 0,Y 440.2,Z 517.811,A -85,B 0,C 180,E1 -9101.978,E2 -9101.978} C_VEL
LIN {X 0,Y 440.75,Z 508.219,A -85,B 0,C 180,E1 -9103.039,E2 -9103.039} C_VEL
LIN {X 0,Y 441.312,Z 496.861,A -85,B 0,C 180,E1 -9104.055,E2 -9104.055} C_VEL
LIN {X 0,Y 441.947,Z 485.467,A -85,B 0,C 180,E1 -9104.858,E2 -9104.858} C_VEL
LIN {X 0,Y 442.531,Z 473.784,A -85,B 0,C 180,E1 -9105.486,E2 -9105.486} C_VEL
LIN {X 0,Y 440.907,Z 461.764,A -85,B 0,C 180,E1 -9106.028,E2 -9106.028} C_VEL
LIN {X 0,Y 438.921,Z 449.56,A -85,B 0,C 180,E1 -9106.453,E2 -9106.453} C_VEL
LIN {X 0,Y 439.267,Z 440.729,A -85,B 0,C 180,E1 -9109.632,E2 -9109.632} C_VEL
LIN {X 0,Y 439.542,Z 432.656,A -85,B 0,C 180,E1 -9112.565,E2 -9112.565} C_VEL
LIN {X 0,Y 440.012,Z 423.372,A -85,B 0,C 180,E1 -9116.054,E2 -9116.054} C_VEL
LIN {X 0,Y 440.393,Z 415.423,A -85,B 0,C 180,E1 -9119.125,E2 -9119.125} C_VEL
LIN {X 0,Y 441.046,Z 406.274,A -85,B 0,C 180,E1 -9122.804,E2 -9122.804} C_VEL
LIN {X 0,Y 441.502,Z 399.311,A -85,B 0,C 180,E1 -9125.724,E2 -9125.724} C_VEL
LIN {X 0,Y 441.265,Z 395.924,A -85,B 0,C 180,E1 -9127.244,E2 -9127.244} C_VEL
LIN {X 0,Y 440.23,Z 390.14,A -85,B 0,C 180,E1 -9129.978,E2 -9129.978} C_VEL
LIN {X 0,Y 439.395,Z 385.755,A -85,B 0,C 180,E1 -9132.203,E2 -9132.203} C_VEL
LIN {X 0,Y 439.397,Z 385.755,A -85,B 0,C 180,E1 -9135.27,E2 -9135.27} C_VEL
LIN {X 0,Y 439.393,Z 385.755,A -85,B 0,C 180,E1 -9138.741,E2 -9138.741} C_VEL
LIN {X 0,Y 439.386,Z 385.756,A -85,B 0,C 180,E1 -9141.604,E2 -9141.604} C_VEL
LIN {X 0,Y 439.395,Z 385.754,A -85,B 0,C 180,E1 -9144.844,E2 -9144.844} C_VEL
LIN {X 0,Y 439.366,Z 385.755,A -85,B 0,C 180,E1 -9148.139,E2 -9148.139} C_VEL
LIN {X 0,Y 439.425,Z 385.749,A -85,B 0,C 180,E1 -9151.598,E2 -9151.598} C_VEL
LIN {X 0,Y 439.398,Z 385.753,A -85,B 0,C 180,E1 -9154.415,E2 -9154.415} C_VEL
LIN {X 0,Y 439.357,Z 385.757,A -85,B 0,C 180,E1 -9157.424,E2 -9157.424} C_VEL
LIN {X 0,Y 439.433,Z 385.751,A -85,B 0,C 180,E1 -9160.662,E2 -9160.662} C_VEL
LIN {X 0,Y 439.453,Z 385.746,A -85,B 0,C 180,E1 -9164.224,E2 -9164.224} C_VEL
LIN {X 0,Y 439.475,Z 385.741,A -85,B 0,C 180,E1 -9168.001,E2 -9168.001} C_VEL
LIN {X 0,Y 439.539,Z 385.734,A -85,B 0,C 180,E1 -9171.726,E2 -9171.726} C_VEL
LIN {X 0,Y 439.612,Z 385.727,A -85,B 0,C 180,E1 -9174.496,E2 -9174.496} C_VEL
LIN {X 0,Y 439.627,Z 385.724,A -85,B 0,C 180,E1 -9178.168,E2 -9178.168} C_VEL
LIN {X 0,Y 439.755,Z 385.708,A -85,B 0,C 180,E1 -9180,E2 -9180} C_VEL
LIN {X 0,Y 439.648,Z 385.723,A -85,B 0,C 180,E1 -9182.749,E2 -9182.749} C_VEL
LIN {X 0,Y 439.609,Z 385.728,A -85,B 0,C 180,E1 -9186.425,E2 -9186.425} C_VEL
LIN {X 0,Y 439.492,Z 385.74,A -85,B 0,C 180,E1 -9189.202,E2 -9189.202} C_VEL
LIN {X 0,Y 439.457,Z 385.745,A -85,B 0,C 180,E1 -9192.938,E2 -9192.938} C_VEL
LIN {X 0,Y 439.439,Z 385.749,A -85,B 0,C 180,E1 -9196.349,E2 -9196.349} C_VEL
LIN {X 0,Y 439.395,Z 385.752,A -85,B 0,C 180,E1 -9199.627,E2 -9199.627} C_VEL
LIN {X 0,Y 439.357,Z 385.76,A -85,B 0,C 180,E1 -9202.576,E2 -9202.576} C_VEL
LIN {X 0,Y 439.398,Z 385.751,A -85,B 0,C 180,E1 -9205.586,E2 -9205.586} C_VEL
LIN {X 0,Y 439.411,Z 385.752,A -85,B 0,C 180,E1 -9208.674,E2 -9208.674} C_VEL
LIN {X 0,Y 439.364,Z 385.758,A -85,B 0,C 180,E1 -9212.031,E2 -9212.031} C_VEL
LIN {X 0,Y 439.391,Z 385.751,A -85,B 0,C 180,E1 -9215.342,E2 -9215.342} C_VEL
LIN {X 0,Y 439.394,Z 385.754,A -85,B 0,C 180,E1 -9218.594,E2 -9218.594} C_VEL
LIN {X 0,Y 439.394,Z 385.752,A -85,B 0,C 180,E1 -9221.259,E2 -9221.259} C_VEL
LIN {X 0,Y 439.397,Z 385.752,A -85,B 0,C 180,E1 -9224.73,E2 -9224.73} C_VEL
LIN {X 0,Y 439.393,Z 385.754,A -85,B 0,C 180,E1 -9227.797,E2 -9227.797} C_VEL
LIN {X 0,Y 439.434,Z 385.75,A -85,B 0,C 180,E1 -9230.229,E2 -9230.229} C_VEL
LIN {X 0,Y 439.375,Z 385.756,A -85,B 0,C 180,E1 -9233.714,E2 -9233.714} C_VEL
LIN {X 0,Y 439.371,Z 385.755,A -85,B 0,C 180,E1 -9237.055,E2 -9237.055} C_VEL
LIN {X 0,Y 439.382,Z 385.756,A -85,B 0,C 180,E1 -9240.275,E2 -9240.275} C_VEL
LIN {X 0,Y 439.429,Z 385.748,A -85,B 0,C 180,E1 -9243.397,E2 -9243.397} C_VEL
LIN {X 0,Y 439.389,Z 385.755,A -85,B 0,C 180,E1 -9246.43,E2 -9246.43} C_VEL
LIN {X 0,Y 439.391,Z 385.754,A -85,B 0,C 180,E1 -9249.398,E2 -9249.398} C_VEL
LIN {X 0,Y 439.433,Z 385.749,A -85,B 0,C 180,E1 -9252.31,E2 -9252.31} C_VEL
LIN {X 0,Y 439.451,Z 385.745,A -85,B 0,C 180,E1 -9255.175,E2 -9255.175} C_VEL
LIN {X 0,Y 439.487,Z 385.743,A -85,B 0,C 180,E1 -9258.002,E2 -9258.002} C_VEL
LIN {X 0,Y 439.551,Z 385.735,A -85,B 0,C 180,E1 -9261.727,E2 -9261.727} C_VEL
LIN {X 0,Y 439.625,Z 385.724,A -85,B 0,C 180,E1 -9264.496,E2 -9264.496} C_VEL
LIN {X 0,Y 439.56,Z 385.735,A -85,B 0,C 180,E1 -9268.168,E2 -9268.168} C_VEL
LIN {X 0,Y 439.326,Z 385.764,A -85,B 0,C 180,E1 -9270,E2 -9270} C_VEL
LIN {X 0,Y 438.923,Z 385.97,A -85,B 0,C 180,E1 -9270.988,E2 -9270.988} C_VEL
LIN {X 0,Y 438.168,Z 386.812,A -85,B 0,C 180,E1 -9271.746,E2 -9271.746} C_VEL
LIN {X 0,Y 435.323,Z 388.36,A -85,B 0,C 180,E1 -9272.975,E2 -9272.975} C_VEL
LIN {X 0,Y 432.958,Z 389.599,A -85,B 0,C 180,E1 -9273.966,E2 -9273.966} C_VEL
LIN {X 0,Y 431.925,Z 390.47,A -85,B 0,C 180,E1 -9274.732,E2 -9274.732} C_VEL
LIN {X 0,Y 431.827,Z 390.741,A -85,B 0,C 180,E1 -9274.992,E2 -9274.992} C_VEL
LIN {X 0,Y 431.767,Z 393.313,A -85,B 0,C 180,E1 -9277.482,E2 -9277.482} C_VEL
LIN {X 0,Y 431.65,Z 397.247,A -85,B 0,C 180,E1 -9281.267,E2 -9281.267} C_VEL
LIN {X 0,Y 431.53,Z 400.335,A -85,B 0,C 180,E1 -9284.14,E2 -9284.14} C_VEL
LIN {X 0,Y 431.519,Z 401.714,A -85,B 0,C 180,E1 -9285.437,E2 -9285.437} C_VEL
LIN {X 0,Y 435.272,Z 417.289,A -85,B 0,C 180,E1 -9286.133,E2 -9286.133} C_VEL
LIN {X 0,Y 435.97,Z 422.189,A -85,B 0,C 180,E1 -9286.388,E2 -9286.388} C_VEL
LIN {X 0,Y 435.432,Z 434.486,A -85,B 0,C 180,E1 -9287.082,E2 -9287.082} C_VEL
LIN {X 0,Y 434.868,Z 445.394,A -85,B 0,C 180,E1 -9287.882,E2 -9287.882} C_VEL
LIN {X 0,Y 434.27,Z 456.27,A -85,B 0,C 180,E1 -9288.885,E2 -9288.885} C_VEL
LIN {X 0,Y 433.67,Z 465.684,A -85,B 0,C 180,E1 -9289.958,E2 -9289.958} C_VEL
LIN {X 0,Y 433.046,Z 474.339,A -85,B 0,C 180,E1 -9291.168,E2 -9291.168} C_VEL
LIN {X 0,Y 432.522,Z 482.251,A -85,B 0,C 180,E1 -9292.528,E2 -9292.528} C_VEL
LIN {X 0,Y 432.092,Z 489.101,A -85,B 0,C 180,E1 -9293.993,E2 -9293.993} C_VEL
LIN {X 0,Y 431.756,Z 494.803,A -85,B 0,C 180,E1 -9295.554,E2 -9295.554} C_VEL
LIN {X 0,Y 431.599,Z 499.102,A -85,B 0,C 180,E1 -9297.125,E2 -9297.125} C_VEL
LIN {X 0,Y 431.379,Z 501.668,A -85,B 0,C 180,E1 -9298.385,E2 -9298.385} C_VEL
LIN {X 0,Y 431.223,Z 504.014,A -85,B 0,C 180,E1 -9300.255,E2 -9300.255} C_VEL
LIN {X 0,Y 431.188,Z 504.804,A -85,B 0,C 180,E1 -9302.053,E2 -9302.053} C_VEL
LIN {X 0,Y 431.244,Z 504.142,A -85,B 0,C 180,E1 -9303.782,E2 -9303.782} C_VEL
LIN {X 0,Y 431.367,Z 502.23,A -85,B 0,C 180,E1 -9305.45,E2 -9305.45} C_VEL
LIN {X 0,Y 431.575,Z 499.128,A -85,B 0,C 180,E1 -9307.065,E2 -9307.065} C_VEL
LIN {X 0,Y 431.828,Z 494.854,A -85,B 0,C 180,E1 -9308.629,E2 -9308.629} C_VEL
LIN {X 0,Y 432.198,Z 489.27,A -85,B 0,C 180,E1 -9310.157,E2 -9310.157} C_VEL
LIN {X 0,Y 432.696,Z 481.776,A -85,B 0,C 180,E1 -9311.753,E2 -9311.753} C_VEL
LIN {X 0,Y 433.266,Z 473.709,A -85,B 0,C 180,E1 -9313.118,E2 -9313.118} C_VEL
LIN {X 0,Y 433.863,Z 464.576,A -85,B 0,C 180,E1 -9314.36,E2 -9314.36} C_VEL
LIN {X 0,Y 434.509,Z 453.955,A -85,B 0,C 180,E1 -9315.528,E2 -9315.528} C_VEL
LIN {X 0,Y 435.074,Z 443.791,A -85,B 0,C 180,E1 -9316.425,E2 -9316.425} C_VEL
LIN {X 0,Y 435.693,Z 431.746,A -85,B 0,C 180,E1 -9317.256,E2 -9317.256} C_VEL
LIN {X 0,Y 435.989,Z 420.424,A -85,B 0,C 180,E1 -9317.859,E2 -9317.859} C_VEL
LIN {X 0,Y 432.889,Z 407.878,A -85,B 0,C 180,E1 -9318.479,E2 -9318.479} C_VEL
LIN {X 0,Y 431.506,Z 402.578,A -85,B 0,C 180,E1 -9318.707,E2 -9318.707} C_VEL
LIN {X 0,Y 431.541,Z 399.495,A -85,B 0,C 180,E1 -9321.767,E2 -9321.767} C_VEL
LIN {X 0,Y 431.641,Z 396.749,A -85,B 0,C 180,E1 -9324.497,E2 -9324.497} C_VEL
LIN {X 0,Y 431.81,Z 393.492,A -85,B 0,C 180,E1 -9327.814,E2 -9327.814} C_VEL
LIN {X 0,Y 431.858,Z 390.586,A -85,B 0,C 180,E1 -9330.776,E2 -9330.776} C_VEL
LIN {X 0,Y 431.955,Z 387.516,A -85,B 0,C 180,E1 -9333.941,E2 -9333.941} C_VEL
LIN {X 0,Y 431.979,Z 386.68,A -85,B 0,C 180,E1 -9334.976,E2 -9334.976} C_VEL
LIN {X 0,Y 432.332,Z 386.637,A -85,B 0,C 180,E1 -9338.044,E2 -9338.044} C_VEL
LIN {X 0,Y 432.382,Z 386.629,A -85,B 0,C 180,E1 -9341.029,E2 -9341.029} C_VEL
LIN {X 0,Y 432.425,Z 386.621,A -85,B 0,C 180,E1 -9343.961,E2 -9343.961} C_VEL
LIN {X 0,Y 432.454,Z 386.619,A -85,B 0,C 180,E1 -9347.803,E2 -9347.803} C_VEL
LIN {X 0,Y 432.487,Z 386.615,A -85,B 0,C 180,E1 -9351.59,E2 -9351.59} C_VEL
LIN {X 0,Y 432.592,Z 386.6,A -85,B 0,C 180,E1 -9354.406,E2 -9354.406} C_VEL
LIN {X 0,Y 432.599,Z 386.601,A -85,B 0,C 180,E1 -9358.138,E2 -9358.138} C_VEL
LIN {X 0,Y 432.727,Z 386.582,A -85,B 0,C 180,E1 -9360,E2 -9360} C_VEL
LIN {X 0,Y 432.599,Z 386.599,A -85,B 0,C 180,E1 -9362.793,E2 -9362.793} C_VEL
LIN {X 0,Y 432.566,Z 386.605,A -85,B 0,C 180,E1 -9366.53,E2 -9366.53} C_VEL
LIN {X 0,Y 432.438,Z 386.62,A -85,B 0,C 180,E1 -9369.353,E2 -9369.353} C_VEL
LIN {X 0,Y 432.425,Z 386.62,A -85,B 0,C 180,E1 -9372.804,E2 -9372.804} C_VEL
LIN {X 0,Y 432.407,Z 386.622,A -85,B 0,C 180,E1 -9376.479,E2 -9376.479} C_VEL
LIN {X 0,Y 432.333,Z 386.634,A -85,B 0,C 180,E1 -9379.961,E2 -9379.961} C_VEL
LIN {X 0,Y 432.314,Z 386.636,A -85,B 0,C 180,E1 -9382.965,E2 -9382.965} C_VEL
LIN {X 0,Y 432.36,Z 386.628,A -85,B 0,C 180,E1 -9386.033,E2 -9386.033} C_VEL
LIN {X 0,Y 432.338,Z 386.631,A -85,B 0,C 180,E1 -9389.188,E2 -9389.188} C_VEL
LIN {X 0,Y 432.318,Z 386.637,A -85,B 0,C 180,E1 -9392.443,E2 -9392.443} C_VEL
LIN {X 0,Y 432.339,Z 386.636,A -85,B 0,C 180,E1 -9395.632,E2 -9395.632} C_VEL
LIN {X 0,Y 432.357,Z 386.632,A -85,B 0,C 180,E1 -9398.718,E2 -9398.718} C_VEL
LIN {X 0,Y 432.363,Z 386.629,A -85,B 0,C 180,E1 -9401.794,E2 -9401.794} C_VEL
LIN {X 0,Y 432.331,Z 386.634,A -85,B 0,C 180,E1 -9404.348,E2 -9404.348} C_VEL
LIN {X 0,Y 432.371,Z 386.732,A -85,B 0,C 180,E1 -9407.412,E2 -9407.412} C_VEL
LIN {X 0,Y 433.325,Z 391.938,A -85,B 0,C 180,E1 -9410.244,E2 -9410.244} C_VEL
LIN {X 0,Y 434.393,Z 397.995,A -85,B 0,C 180,E1 -9413.23,E2 -9413.23} C_VEL
LIN {X 0,Y 434.343,Z 401.778,A -85,B 0,C 180,E1 -9414.942,E2 -9414.942} C_VEL
LIN {X 0,Y 433.832,Z 408.152,A -85,B 0,C 180,E1 -9417.684,E2 -9417.684} C_VEL
LIN {X 0,Y 433.3,Z 415.92,A -85,B 0,C 180,E1 -9420.884,E2 -9420.884} C_VEL
LIN {X 0,Y 432.849,Z 423.846,A -85,B 0,C 180,E1 -9423.999,E2 -9423.999} C_VEL
LIN {X 0,Y 432.427,Z 433.059,A -85,B 0,C 180,E1 -9427.521,E2 -9427.521} C_VEL
LIN {X 0,Y 432.104,Z 442.533,A -85,B 0,C 180,E1 -9431.017,E2 -9431.017} C_VEL
LIN {X 0,Y 431.848,Z 448.965,A -85,B 0,C 180,E1 -9433.297,E2 -9433.297} C_VEL
LIN {X 0,Y 434.003,Z 462.689,A -85,B 0,C 180,E1 -9433.764,E2 -9433.764} C_VEL
LIN {X 0,Y 435.598,Z 474.318,A -85,B 0,C 180,E1 -9434.321,E2 -9434.321} C_VEL
LIN {X 0,Y 434.968,Z 486.563,A -85,B 0,C 180,E1 -9435.018,E2 -9435.018} C_VEL
LIN {X 0,Y 434.232,Z 499.069,A -85,B 0,C 180,E1 -9435.95,E2 -9435.95} C_VEL
LIN {X 0,Y 433.624,Z 510.056,A -85,B 0,C 180,E1 -9437.004,E2 -9437.004} C_VEL
LIN {X 0,Y 433.078,Z 519.021,A -85,B 0,C 180,E1 -9438.059,E2 -9438.059} C_VEL
LIN {X 0,Y 432.402,Z 528.766,A -85,B 0,C 180,E1 -9439.464,E2 -9439.464} C_VEL
LIN {X 0,Y 431.95,Z 536.538,A -85,B 0,C 180,E1 -9440.872,E2 -9440.872} C_VEL
LIN {X 0,Y 431.549,Z 543.707,A -85,B 0,C 180,E1 -9442.514,E2 -9442.514} C_VEL
LIN {X 0,Y 431.378,Z 548.429,A -85,B 0,C 180,E1 -9443.903,E2 -9443.903} C_VEL
LIN {X 0,Y 431.29,Z 552.141,A -85,B 0,C 180,E1 -9445.326,E2 -9445.326} C_VEL
LIN {X 0,Y 431.211,Z 554.027,A -85,B 0,C 180,E1 -9446.262,E2 -9446.262} C_VEL
LIN {X 0,Y 431.28,Z 555.448,A -85,B 0,C 180,E1 -9447.198,E2 -9447.198} C_VEL
LIN {X 0,Y 431.198,Z 557.078,A -85,B 0,C 180,E1 -9449.066,E2 -9449.066} C_VEL
LIN {X 0,Y 431.216,Z 557.303,A -85,B 0,C 180,E1 -9450,E2 -9450} C_VEL
LIN {X 0,Y 431.198,Z 557.087,A -85,B 0,C 180,E1 -9450.934,E2 -9450.934} C_VEL
LIN {X 0,Y 431.28,Z 555.482,A -85,B 0,C 180,E1 -9452.802,E2 -9452.802} C_VEL
LIN {X 0,Y 431.21,Z 554.071,A -85,B 0,C 180,E1 -9453.738,E2 -9453.738} C_VEL
LIN {X 0,Y 431.368,Z 551.119,A -85,B 0,C 180,E1 -9455.141,E2 -9455.141} C_VEL
LIN {X 0,Y 431.441,Z 547.113,A -85,B 0,C 180,E1 -9456.547,E2 -9456.547} C_VEL
LIN {X 0,Y 431.711,Z 540.958,A -85,B 0,C 180,E1 -9458.189,E2 -9458.189} C_VEL
LIN {X 0,Y 432.103,Z 534.241,A -85,B 0,C 180,E1 -9459.596,E2 -9459.596} C_VEL
LIN {X 0,Y 432.557,Z 525.91,A -85,B 0,C 180,E1 -9461.005,E2 -9461.005} C_VEL
LIN {X 0,Y 433.225,Z 517.383,A -85,B 0,C 180,E1 -9462.174,E2 -9462.174} C_VEL
LIN {X 0,Y 433.818,Z 507.383,A -85,B 0,C 180,E1 -9463.293,E2 -9463.293} C_VEL
LIN {X 0,Y 434.388,Z 496.433,A -85,B 0,C 180,E1 -9464.284,E2 -9464.284} C_VEL
LIN {X 0,Y 435.082,Z 485.042,A -85,B 0,C 180,E1 -9465.097,E2 -9465.097} C_VEL
LIN {X 0,Y 435.564,Z 473.351,A -85,B 0,C 180,E1 -9465.74,E2 -9465.74} C_VEL
LIN {X 0,Y 433.723,Z 460.968,A -85,B 0,C 180,E1 -9466.313,E2 -9466.313} C_VEL
LIN {X 0,Y 431.851,Z 449.167,A -85,B 0,C 180,E1 -9466.721,E2 -9466.721} C_VEL
LIN {X 0,Y 432.197,Z 440.302,A -85,B 0,C 180,E1 -9469.967,E2 -9469.967} C_VEL
LIN {X 0,Y 432.507,Z 432.325,A -85,B 0,C 180,E1 -9472.953,E2 -9472.953} C_VEL
LIN {X 0,Y 433.01,Z 423.355,A -85,B 0,C 180,E1 -9476.394,E2 -9476.394} C_VEL
LIN {X 0,Y 433.417,Z 415.162,A -85,B 0,C 180,E1 -9479.64,E2 -9479.64} C_VEL
LIN {X 0,Y 433.982,Z 407.839,A -85,B 0,C 180,E1 -9482.637,E2 -9482.637} C_VEL
LIN {X 0,Y 434.496,Z 400.888,A -85,B 0,C 180,E1 -9485.612,E2 -9485.612} C_VEL
LIN {X 0,Y 434.454,Z 398.296,A -85,B 0,C 180,E1 -9486.764,E2 -9486.764} C_VEL
LIN {X 0,Y 433.357,Z 392.048,A -85,B 0,C 180,E1 -9489.755,E2 -9489.755} C_VEL
LIN {X 0,Y 432.353,Z 386.632,A -85,B 0,C 180,E1 -9492.579,E2 -9492.579} C_VEL
LIN {X 0,Y 432.328,Z 386.635,A -85,B 0,C 180,E1 -9495.664,E2 -9495.664} C_VEL
LIN {X 0,Y 432.361,Z 386.631,A -85,B 0,C 180,E1 -9498.392,E2 -9498.392} C_VEL
LIN {X 0,Y 432.347,Z 386.633,A -85,B 0,C 180,E1 -9501.851,E2 -9501.851} C_VEL
LIN {X 0,Y 432.334,Z 386.633,A -85,B 0,C 180,E1 -9505.322,E2 -9505.322} C_VEL
LIN {X 0,Y 432.314,Z 386.637,A -85,B 0,C 180,E1 -9508.653,E2 -9508.653} C_VEL
LIN {X 0,Y 432.375,Z 386.626,A -85,B 0,C 180,E1 -9511.876,E2 -9511.876} C_VEL
LIN {X 0,Y 432.344,Z 386.633,A -85,B 0,C 180,E1 -9514.998,E2 -9514.998} C_VEL
LIN {X 0,Y 432.349,Z 386.628,A -85,B 0,C 180,E1 -9518.045,E2 -9518.045} C_VEL
LIN {X 0,Y 432.378,Z 386.628,A -85,B 0,C 180,E1 -9521.029,E2 -9521.029} C_VEL
LIN {X 0,Y 432.422,Z 386.62,A -85,B 0,C 180,E1 -9523.961,E2 -9523.961} C_VEL
LIN {X 0,Y 432.451,Z 386.615,A -85,B 0,C 180,E1 -9527.803,E2 -9527.803} C_VEL
LIN {X 0,Y 432.483,Z 386.613,A -85,B 0,C 180,E1 -9531.59,E2 -9531.59} C_VEL
LIN {X 0,Y 432.588,Z 386.602,A -85,B 0,C 180,E1 -9534.406,E2 -9534.406} C_VEL
LIN {X 0,Y 432.597,Z 386.599,A -85,B 0,C 180,E1 -9538.138,E2 -9538.138} C_VEL
LIN {X 0,Y 432.725,Z 386.583,A -85,B 0,C 180,E1 -9540,E2 -9540} C_VEL
LIN {X 0,Y 432.597,Z 386.601,A -85,B 0,C 180,E1 -9542.794,E2 -9542.794} C_VEL
LIN {X 0,Y 432.564,Z 386.605,A -85,B 0,C 180,E1 -9546.531,E2 -9546.531} C_VEL
LIN {X 0,Y 432.435,Z 386.619,A -85,B 0,C 180,E1 -9549.353,E2 -9549.353} C_VEL
LIN {X 0,Y 432.422,Z 386.622,A -85,B 0,C 180,E1 -9552.804,E2 -9552.804} C_VEL
LIN {X 0,Y 432.404,Z 386.625,A -85,B 0,C 180,E1 -9556.479,E2 -9556.479} C_VEL
LIN {X 0,Y 432.331,Z 386.633,A -85,B 0,C 180,E1 -9559.961,E2 -9559.961} C_VEL
LIN {X 0,Y 432.312,Z 386.635,A -85,B 0,C 180,E1 -9562.965,E2 -9562.965} C_VEL
LIN {X 0,Y 432.358,Z 386.631,A -85,B 0,C 180,E1 -9566.033,E2 -9566.033} C_VEL
LIN {X 0,Y 432.336,Z 386.631,A -85,B 0,C 180,E1 -9569.188,E2 -9569.188} C_VEL
LIN {X 0,Y 432.317,Z 386.637,A -85,B 0,C 180,E1 -9572.444,E2 -9572.444} C_VEL
LIN {X 0,Y 432.34,Z 386.63,A -85,B 0,C 180,E1 -9575.633,E2 -9575.633} C_VEL
LIN {X 0,Y 432.356,Z 386.63,A -85,B 0,C 180,E1 -9578.719,E2 -9578.719} C_VEL
LIN {X 0,Y 432.361,Z 386.63,A -85,B 0,C 180,E1 -9581.794,E2 -9581.794} C_VEL
LIN {X 0,Y 432.33,Z 386.635,A -85,B 0,C 180,E1 -9584.348,E2 -9584.348} C_VEL
LIN {X 0,Y 432.317,Z 386.633,A -85,B 0,C 180,E1 -9587.017,E2 -9587.017} C_VEL
LIN {X 0,Y 432.339,Z 386.633,A -85,B 0,C 180,E1 -9589.82,E2 -9589.82} C_VEL
LIN {X 0,Y 432.314,Z 386.633,A -85,B 0,C 180,E1 -9593.024,E2 -9593.024} C_VEL
LIN {X 0,Y 432.359,Z 386.632,A -85,B 0,C 180,E1 -9595.997,E2 -9595.997} C_VEL
LIN {X 0,Y 432.347,Z 386.631,A -85,B 0,C 180,E1 -9599.49,E2 -9599.49} C_VEL
LIN {X 0,Y 432.392,Z 386.623,A -85,B 0,C 180,E1 -9602.929,E2 -9602.929} C_VEL
LIN {X 0,Y 432.373,Z 386.629,A -85,B 0,C 180,E1 -9606.024,E2 -9606.024} C_VEL
LIN {X 0,Y 432.352,Z 386.629,A -85,B 0,C 180,E1 -9609.047,E2 -9609.047} C_VEL
LIN {X 0,Y 432.38,Z 386.628,A -85,B 0,C 180,E1 -9612.012,E2 -9612.012} C_VEL
LIN {X 0,Y 432.398,Z 386.623,A -85,B 0,C 180,E1 -9614.927,E2 -9614.927} C_VEL
LIN {X 0,Y 432.462,Z 386.618,A -85,B 0,C 180,E1 -9617.804,E2 -9617.804} C_VEL
LIN {X 0,Y 432.495,Z 386.614,A -85,B 0,C 180,E1 -9621.591,E2 -9621.591} C_VEL
LIN {X 0,Y 432.602,Z 386.599,A -85,B 0,C 180,E1 -9624.407,E2 -9624.407} C_VEL
LIN {X 0,Y 432.532,Z 386.61,A -85,B 0,C 180,E1 -9628.138,E2 -9628.138} C_VEL
LIN {X 0,Y 432.29,Z 386.641,A -85,B 0,C 180,E1 -9630,E2 -9630} C_VEL
LIN {X 0,Y 431.869,Z 386.719,A -85,B 0,C 180,E1 -9630.951,E2 -9630.951} C_VEL
LIN {X 0,Y 431.861,Z 390.412,A -85,B 0,C 180,E1 -9634.667,E2 -9634.667} C_VEL
LIN {X 0,Y 431.827,Z 390.741,A -85,B 0,C 180,E1 -9634.992,E2 -9634.992} C_VEL
LIN {X 0,Y 431.115,Z 391.603,A -85,B 0,C 180,E1 -9635.762,E2 -9635.762} C_VEL
LIN {X 0,Y 428.209,Z 393.2,A -85,B 0,C 180,E1 -9637.009,E2 -9637.009} C_VEL
LIN {X 0,Y 425.76,Z 394.501,A -85,B 0,C 180,E1 -9638.015,E2 -9638.015} C_VEL
LIN {X 0,Y 424.695,Z 395.409,A -85,B 0,C 180,E1 -9638.795,E2 -9638.795} C_VEL
LIN {X 0,Y 424.6,Z 395.691,A -85,B 0,C 180,E1 -9639.06,E2 -9639.06} C_VEL
LIN {X 0,Y 424.558,Z 399.171,A -85,B 0,C 180,E1 -9642.427,E2 -9642.427} C_VEL
LIN {X 0,Y 424.491,Z 402.073,A -85,B 0,C 180,E1 -9645.177,E2 -9645.177} C_VEL
LIN {X 0,Y 427.862,Z 415.966,A -85,B 0,C 180,E1 -9645.786,E2 -9645.786} C_VEL
LIN {X 0,Y 429.123,Z 423.101,A -85,B 0,C 180,E1 -9646.166,E2 -9646.166} C_VEL
LIN {X 0,Y 428.542,Z 436.034,A -85,B 0,C 180,E1 -9646.923,E2 -9646.923} C_VEL
LIN {X 0,Y 427.947,Z 446.627,A -85,B 0,C 180,E1 -9647.727,E2 -9647.727} C_VEL
LIN {X 0,Y 427.36,Z 456.943,A -85,B 0,C 180,E1 -9648.704,E2 -9648.704} C_VEL
LIN {X 0,Y 426.708,Z 466.671,A -85,B 0,C 180,E1 -9649.843,E2 -9649.843} C_VEL
LIN {X 0,Y 426.053,Z 474.939,A -85,B 0,C 180,E1 -9651.025,E2 -9651.025} C_VEL
LIN {X 0,Y 425.457,Z 483.605,A -85,B 0,C 180,E1 -9652.559,E2 -9652.559} C_VEL
LIN {X 0,Y 425.048,Z 489.651,A -85,B 0,C 180,E1 -9653.897,E2 -9653.897} C_VEL
LIN {X 0,Y 424.694,Z 495.319,A -85,B 0,C 180,E1 -9655.484,E2 -9655.484} C_VEL
LIN {X 0,Y 424.524,Z 499.602,A -85,B 0,C 180,E1 -9657.083,E2 -9657.083} C_VEL
LIN {X 0,Y 424.268,Z 502.678,A -85,B 0,C 180,E1 -9658.71,E2 -9658.71} C_VEL
LIN {X 0,Y 424.14,Z 504.671,A -85,B 0,C 180,E1 -9660.498,E2 -9660.498} C_VEL
LIN {X 0,Y 424.113,Z 505.206,A -85,B 0,C 180,E1 -9662.314,E2 -9662.314} C_VEL
LIN {X 0,Y 424.177,Z 504.38,A -85,B 0,C 180,E1 -9664.062,E2 -9664.062} C_VEL
LIN {X 0,Y 424.325,Z 502.316,A -85,B 0,C 180,E1 -9665.749,E2 -9665.749} C_VEL
LIN {X 0,Y 424.558,Z 499.041,A -85,B 0,C 180,E1 -9667.384,E2 -9667.384} C_VEL
LIN {X 0,Y 424.853,Z 494.552,A -85,B 0,C 180,E1 -9668.969,E2 -9668.969} C_VEL
LIN {X 0,Y 425.229,Z 488.819,A -85,B 0,C 180,E1 -9670.512,E2 -9670.512} C_VEL
LIN {X 0,Y 425.765,Z 481.657,A -85,B 0,C 180,E1 -9672.029,E2 -9672.029} C_VEL
LIN {X 0,Y 426.381,Z 472.777,A -85,B 0,C 180,E1 -9673.51,E2 -9673.51} C_VEL
LIN {X 0,Y 427.012,Z 464.055,A -85,B 0,C 180,E1 -9674.686,E2 -9674.686} C_VEL
LIN {X 0,Y 427.663,Z 453.945,A -85,B 0,C 180,E1 -9675.799,E2 -9675.799} C_VEL
LIN {X 0,Y 428.288,Z 442.984,A -85,B 0,C 180,E1 -9676.761,E2 -9676.761} C_VEL
LIN {X 0,Y 428.93,Z 430.871,A -85,B 0,C 180,E1 -9677.589,E2 -9677.589} C_VEL
LIN {X 0,Y 429.31,Z 422.794,A -85,B 0,C 180,E1 -9678.024,E2 -9678.024} C_VEL
LIN {X 0,Y 426.549,Z 410.787,A -85,B 0,C 180,E1 -9678.651,E2 -9678.651} C_VEL
LIN {X 0,Y 424.498,Z 403.021,A -85,B 0,C 180,E1 -9679.009,E2 -9679.009} C_VEL
LIN {X 0,Y 424.516,Z 399.41,A -85,B 0,C 180,E1 -9682.622,E2 -9682.622} C_VEL
LIN {X 0,Y 424.655,Z 396.235,A -85,B 0,C 180,E1 -9685.841,E2 -9685.841} C_VEL
LIN {X 0,Y 424.789,Z 393.036,A -85,B 0,C 180,E1 -9689.144,E2 -9689.144} C_VEL
LIN {X 0,Y 424.84,Z 389.88,A -85,B 0,C 180,E1 -9692.406,E2 -9692.406} C_VEL
LIN {X 0,Y 424.908,Z 387.865,A -85,B 0,C 180,E1 -9694.53,E2 -9694.53} C_VEL
LIN {X 0,Y 425.145,Z 387.533,A -85,B 0,C 180,E1 -9696.625,E2 -9696.625} C_VEL
LIN {X 0,Y 425.29,Z 387.514,A -85,B 0,C 180,E1 -9699.694,E2 -9699.694} C_VEL
LIN {X 0,Y 425.337,Z 387.504,A -85,B 0,C 180,E1 -9702.697,E2 -9702.697} C_VEL
LIN {X 0,Y 425.342,Z 387.505,A -85,B 0,C 180,E1 -9705.65,E2 -9705.65} C_VEL
LIN {X 0,Y 425.348,Z 387.503,A -85,B 0,C 180,E1 -9708.564,E2 -9708.564} C_VEL
LIN {X 0,Y 425.533,Z 387.478,A -85,B 0,C 180,E1 -9712.407,E2 -9712.407} C_VEL
LIN {X 0,Y 425.548,Z 387.478,A -85,B 0,C 180,E1 -9714.313,E2 -9714.313} C_VEL
LIN {X 0,Y 425.569,Z 387.477,A -85,B 0,C 180,E1 -9718.107,E2 -9718.107} C_VEL
LIN {X 0,Y 425.696,Z 387.457,A -85,B 0,C 180,E1 -9720,E2 -9720} C_VEL
LIN {X 0,Y 425.551,Z 387.477,A -85,B 0,C 180,E1 -9722.84,E2 -9722.84} C_VEL
LIN {X 0,Y 425.523,Z 387.482,A -85,B 0,C 180,E1 -9726.639,E2 -9726.639} C_VEL
LIN {X 0,Y 425.396,Z 387.497,A -85,B 0,C 180,E1 -9729.509,E2 -9729.509} C_VEL
LIN {X 0,Y 425.388,Z 387.496,A -85,B 0,C 180,E1 -9732.904,E2 -9732.904} C_VEL
LIN {X 0,Y 425.356,Z 387.5,A -85,B 0,C 180,E1 -9736.605,E2 -9736.605} C_VEL
LIN {X 0,Y 425.323,Z 387.505,A -85,B 0,C 180,E1 -9739.636,E2 -9739.636} C_VEL
LIN {X 0,Y 425.302,Z 387.51,A -85,B 0,C 180,E1 -9743.365,E2 -9743.365} C_VEL
LIN {X 0,Y 425.344,Z 387.502,A -85,B 0,C 180,E1 -9746.845,E2 -9746.845} C_VEL
LIN {X 0,Y 425.286,Z 387.513,A -85,B 0,C 180,E1 -9749.72,E2 -9749.72} C_VEL
LIN {X 0,Y 425.277,Z 387.514,A -85,B 0,C 180,E1 -9753.048,E2 -9753.048} C_VEL
LIN {X 0,Y 425.279,Z 387.515,A -85,B 0,C 180,E1 -9755.929,E2 -9755.929} C_VEL
LIN {X 0,Y 425.31,Z 387.51,A -85,B 0,C 180,E1 -9759.046,E2 -9759.046} C_VEL
LIN {X 0,Y 425.312,Z 387.508,A -85,B 0,C 180,E1 -9761.962,E2 -9761.962} C_VEL
LIN {X 0,Y 425.283,Z 387.514,A -85,B 0,C 180,E1 -9765.284,E2 -9765.284} C_VEL
LIN {X 0,Y 425.305,Z 387.575,A -85,B 0,C 180,E1 -9767.005,E2 -9767.005} C_VEL
LIN {X 0,Y 426.291,Z 392.934,A -85,B 0,C 180,E1 -9769.987,E2 -9769.987} C_VEL
LIN {X 0,Y 427.375,Z 399.078,A -85,B 0,C 180,E1 -9773.115,E2 -9773.115} C_VEL
LIN {X 0,Y 427.377,Z 402.853,A -85,B 0,C 180,E1 -9774.862,E2 -9774.862} C_VEL
LIN {X 0,Y 426.824,Z 409.197,A -85,B 0,C 180,E1 -9777.647,E2 -9777.647} C_VEL
LIN {X 0,Y 426.27,Z 416.968,A -85,B 0,C 180,E1 -9780.906,E2 -9780.906} C_VEL
LIN {X 0,Y 425.785,Z 424.848,A -85,B 0,C 180,E1 -9784.062,E2 -9784.062} C_VEL
LIN {X 0,Y 425.399,Z 432.772,A -85,B 0,C 180,E1 -9787.155,E2 -9787.155} C_VEL
LIN {X 0,Y 425.081,Z 442.123,A -85,B 0,C 180,E1 -9790.691,E2 -9790.691} C_VEL
LIN {X 0,Y 424.772,Z 448.34,A -85,B 0,C 180,E1 -9792.993,E2 -9792.993} C_VEL
LIN {X 0,Y 427.05,Z 463.175,A -85,B 0,C 180,E1 -9793.529,E2 -9793.529} C_VEL
LIN {X 0,Y 428.679,Z 474.976,A -85,B 0,C 180,E1 -9794.122,E2 -9794.122} C_VEL
LIN {X 0,Y 427.973,Z 487.86,A -85,B 0,C 180,E1 -9794.889,E2 -9794.889} C_VEL
LIN {X 0,Y 427.242,Z 499.616,A -85,B 0,C 180,E1 -9795.807,E2 -9795.807} C_VEL
LIN {X 0,Y 426.592,Z 510.669,A -85,B 0,C 180,E1 -9796.907,E2 -9796.907} C_VEL
LIN {X 0,Y 425.936,Z 520.357,A -85,B 0,C 180,E1 -9798.097,E2 -9798.097} C_VEL
LIN {X 0,Y 425.381,Z 528.309,A -85,B 0,C 180,E1 -9799.288,E2 -9799.288} C_VEL
LIN {X 0,Y 424.899,Z 536.086,A -85,B 0,C 180,E1 -9800.719,E2 -9800.719} C_VEL
LIN {X 0,Y 424.465,Z 543.259,A -85,B 0,C 180,E1 -9802.388,E2 -9802.388} C_VEL
LIN {X 0,Y 424.278,Z 548.421,A -85,B 0,C 180,E1 -9803.944,E2 -9803.944} C_VEL
LIN {X 0,Y 424.226,Z 551.704,A -85,B 0,C 180,E1 -9805.248,E2 -9805.248} C_VEL
LIN {X 0,Y 424.121,Z 553.59,A -85,B 0,C 180,E1 -9806.199,E2 -9806.199} C_VEL
LIN {X 0,Y 424.192,Z 555.014,A -85,B 0,C 180,E1 -9807.151,E2 -9807.151} C_VEL
LIN {X 0,Y 424.115,Z 556.648,A -85,B 0,C 180,E1 -9809.05,E2 -9809.05} C_VEL
LIN {X 0,Y 424.13,Z 556.874,A -85,B 0,C 180,E1 -9810,E2 -9810} C_VEL
LIN {X 0,Y 424.115,Z 556.659,A -85,B 0,C 180,E1 -9810.949,E2 -9810.949} C_VEL
LIN {X 0,Y 424.192,Z 555.056,A -85,B 0,C 180,E1 -9812.849,E2 -9812.849} C_VEL
LIN {X 0,Y 424.12,Z 553.644,A -85,B 0,C 180,E1 -9813.8,E2 -9813.8} C_VEL
LIN {X 0,Y 424.279,Z 550.693,A -85,B 0,C 180,E1 -9815.227,E2 -9815.227} C_VEL
LIN {X 0,Y 424.359,Z 546.686,A -85,B 0,C 180,E1 -9816.657,E2 -9816.657} C_VEL
LIN {X 0,Y 424.651,Z 540.531,A -85,B 0,C 180,E1 -9818.326,E2 -9818.326} C_VEL
LIN {X 0,Y 425.047,Z 533.812,A -85,B 0,C 180,E1 -9819.757,E2 -9819.757} C_VEL
LIN {X 0,Y 425.555,Z 525.482,A -85,B 0,C 180,E1 -9821.189,E2 -9821.189} C_VEL
LIN {X 0,Y 426.247,Z 516.954,A -85,B 0,C 180,E1 -9822.377,E2 -9822.377} C_VEL
LIN {X 0,Y 426.835,Z 507.464,A -85,B 0,C 180,E1 -9823.462,E2 -9823.462} C_VEL
LIN {X 0,Y 427.476,Z 496.005,A -85,B 0,C 180,E1 -9824.52,E2 -9824.52} C_VEL
LIN {X 0,Y 428.206,Z 484.615,A -85,B 0,C 180,E1 -9825.346,E2 -9825.346} C_VEL
LIN {X 0,Y 428.678,Z 474.152,A -85,B 0,C 180,E1 -9825.938,E2 -9825.938} C_VEL
LIN {X 0,Y 426.721,Z 460.653,A -85,B 0,C 180,E1 -9826.584,E2 -9826.584} C_VEL
LIN {X 0,Y 424.79,Z 448.748,A -85,B 0,C 180,E1 -9827.007,E2 -9827.007} C_VEL
LIN {X 0,Y 425.117,Z 441.089,A -85,B 0,C 180,E1 -9829.876,E2 -9829.876} C_VEL
LIN {X 0,Y 425.424,Z 433.337,A -85,B 0,C 180,E1 -9832.843,E2 -9832.843} C_VEL
LIN {X 0,Y 425.866,Z 425.391,A -85,B 0,C 180,E1 -9835.932,E2 -9835.932} C_VEL
LIN {X 0,Y 426.349,Z 417.491,A -85,B 0,C 180,E1 -9839.113,E2 -9839.113} C_VEL
LIN {X 0,Y 427.012,Z 408.344,A -85,B 0,C 180,E1 -9842.924,E2 -9842.924} C_VEL
LIN {X 0,Y 427.525,Z 401.961,A -85,B 0,C 180,E1 -9845.701,E2 -9845.701} C_VEL
LIN {X 0,Y 427.227,Z 398.097,A -85,B 0,C 180,E1 -9847.491,E2 -9847.491} C_VEL
LIN {X 0,Y 426.077,Z 391.693,A -85,B 0,C 180,E1 -9850.645,E2 -9850.645} C_VEL
LIN {X 0,Y 425.287,Z 387.512,A -85,B 0,C 180,E1 -9852.934,E2 -9852.934} C_VEL
LIN {X 0,Y 425.257,Z 387.516,A -85,B 0,C 180,E1 -9856.043,E2 -9856.043} C_VEL
LIN {X 0,Y 425.299,Z 387.51,A -85,B 0,C 180,E1 -9858.624,E2 -9858.624} C_VEL
LIN {X 0,Y 425.318,Z 387.508,A -85,B 0,C 180,E1 -9861.103,E2 -9861.103} C_VEL
LIN {X 0,Y 425.294,Z 387.51,A -85,B 0,C 180,E1 -9864.664,E2 -9864.664} C_VEL
LIN {X 0,Y 425.258,Z 387.512,A -85,B 0,C 180,E1 -9868.072,E2 -9868.072} C_VEL
LIN {X 0,Y 425.324,Z 387.506,A -85,B 0,C 180,E1 -9871.367,E2 -9871.367} C_VEL
LIN {X 0,Y 425.288,Z 387.511,A -85,B 0,C 180,E1 -9874.554,E2 -9874.554} C_VEL
LIN {X 0,Y 425.28,Z 387.509,A -85,B 0,C 180,E1 -9877.661,E2 -9877.661} C_VEL
LIN {X 0,Y 425.354,Z 387.504,A -85,B 0,C 180,E1 -9880.704,E2 -9880.704} C_VEL
LIN {X 0,Y 425.38,Z 387.497,A -85,B 0,C 180,E1 -9883.688,E2 -9883.688} C_VEL
LIN {X 0,Y 425.403,Z 387.493,A -85,B 0,C 180,E1 -9887.598,E2 -9887.598} C_VEL
LIN {X 0,Y 425.434,Z 387.491,A -85,B 0,C 180,E1 -9891.45,E2 -9891.45} C_VEL
LIN {X 0,Y 425.545,Z 387.479,A -85,B 0,C 180,E1 -9894.313,E2 -9894.313} C_VEL
LIN {X 0,Y 425.567,Z 387.475,A -85,B 0,C 180,E1 -9898.107,E2 -9898.107} C_VEL
LIN {X 0,Y 425.695,Z 387.459,A -85,B 0,C 180,E1 -9900,E2 -9900} C_VEL
LIN {X 0,Y 425.549,Z 387.479,A -85,B 0,C 180,E1 -9902.84,E2 -9902.84} C_VEL
LIN {X 0,Y 425.522,Z 387.483,A -85,B 0,C 180,E1 -9906.639,E2 -9906.639} C_VEL
LIN {X 0,Y 425.394,Z 387.495,A -85,B 0,C 180,E1 -9909.51,E2 -9909.51} C_VEL
LIN {X 0,Y 425.385,Z 387.498,A -85,B 0,C 180,E1 -9912.904,E2 -9912.904} C_VEL
LIN {X 0,Y 425.353,Z 387.504,A -85,B 0,C 180,E1 -9916.605,E2 -9916.605} C_VEL
LIN {X 0,Y 425.321,Z 387.505,A -85,B 0,C 180,E1 -9919.636,E2 -9919.636} C_VEL
LIN {X 0,Y 425.299,Z 387.507,A -85,B 0,C 180,E1 -9923.366,E2 -9923.366} C_VEL
LIN {X 0,Y 425.342,Z 387.504,A -85,B 0,C 180,E1 -9926.845,E2 -9926.845} C_VEL
LIN {X 0,Y 425.284,Z 387.51,A -85,B 0,C 180,E1 -9929.72,E2 -9929.72} C_VEL
LIN {X 0,Y 425.276,Z 387.51,A -85,B 0,C 180,E1 -9933.049,E2 -9933.049} C_VEL
LIN {X 0,Y 425.28,Z 387.512,A -85,B 0,C 180,E1 -9935.93,E2 -9935.93} C_VEL
LIN {X 0,Y 425.309,Z 387.506,A -85,B 0,C 180,E1 -9939.047,E2 -9939.047} C_VEL
LIN {X 0,Y 425.311,Z 387.509,A -85,B 0,C 180,E1 -9941.963,E2 -9941.963} C_VEL
LIN {X 0,Y 425.281,Z 387.509,A -85,B 0,C 180,E1 -9945.284,E2 -9945.284} C_VEL
LIN {X 0,Y 425.272,Z 387.513,A -85,B 0,C 180,E1 -9948.622,E2 -9948.622} C_VEL
LIN {X 0,Y 425.313,Z 387.505,A -85,B 0,C 180,E1 -9951.104,E2 -9951.104} C_VEL
LIN {X 0,Y 425.299,Z 387.508,A -85,B 0,C 180,E1 -9954.665,E2 -9954.665} C_VEL
LIN {X 0,Y 425.265,Z 387.515,A -85,B 0,C 180,E1 -9958.074,E2 -9958.074} C_VEL
LIN {X 0,Y 425.331,Z 387.504,A -85,B 0,C 180,E1 -9961.369,E2 -9961.369} C_VEL
LIN {X 0,Y 425.297,Z 387.509,A -85,B 0,C 180,E1 -9964.556,E2 -9964.556} C_VEL
LIN {X 0,Y 425.29,Z 387.511,A -85,B 0,C 180,E1 -9967.662,E2 -9967.662} C_VEL
LIN {X 0,Y 425.364,Z 387.499,A -85,B 0,C 180,E1 -9970.705,E2 -9970.705} C_VEL
LIN {X 0,Y 425.391,Z 387.499,A -85,B 0,C 180,E1 -9973.689,E2 -9973.689} C_VEL
LIN {X 0,Y 425.415,Z 387.495,A -85,B 0,C 180,E1 -9977.599,E2 -9977.599} C_VEL
LIN {X 0,Y 425.446,Z 387.491,A -85,B 0,C 180,E1 -9981.45,E2 -9981.45} C_VEL
LIN {X 0,Y 425.558,Z 387.476,A -85,B 0,C 180,E1 -9984.314,E2 -9984.314} C_VEL
LIN {X 0,Y 425.502,Z 387.486,A -85,B 0,C 180,E1 -9988.107,E2 -9988.107} C_VEL
LIN {X 0,Y 425.254,Z 387.517,A -85,B 0,C 180,E1 -9990,E2 -9990} C_VEL
LIN {X 0,Y 424.816,Z 387.573,A -85,B 0,C 180,E1 -9990.948,E2 -9990.948} C_VEL
LIN {X 0,Y 424.805,Z 391.267,A -85,B 0,C 180,E1 -9994.745,E2 -9994.745} C_VEL
LIN {X 0,Y 424.7,Z 394.198,A -85,B 0,C 180,E1 -9997.608,E2 -9997.608} C_VEL
LIN {X 0,Y 424.6,Z 395.691,A -85,B 0,C 180,E1 -9999.06,E2 -9999.06} C_VEL
LIN {X 0,Y 423.904,Z 396.571,A -85,B 0,C 180,E1 -9999.843,E2 -9999.843} C_VEL
LIN {X 0,Y 421.018,Z 398.179,A -85,B 0,C 180,E1 -10001.112,E2 -10001.112} C_VEL
LIN {X 0,Y 418.578,Z 399.486,A -85,B 0,C 180,E1 -10002.135,E2 -10002.135} C_VEL
LIN {X 0,Y 417.518,Z 400.422,A -85,B 0,C 180,E1 -10002.928,E2 -10002.928} C_VEL
LIN {X 0,Y 417.424,Z 400.714,A -85,B 0,C 180,E1 -10003.197,E2 -10003.197} C_VEL
LIN {X 0,Y 417.43,Z 402.46,A -85,B 0,C 180,E1 -10004.877,E2 -10004.877} C_VEL
LIN {X 0,Y 421.017,Z 417.086,A -85,B 0,C 180,E1 -10005.553,E2 -10005.553} C_VEL
LIN {X 0,Y 422.304,Z 423.996,A -85,B 0,C 180,E1 -10005.938,E2 -10005.938} C_VEL
LIN {X 0,Y 421.661,Z 436.859,A -85,B 0,C 180,E1 -10006.709,E2 -10006.709} C_VEL
LIN {X 0,Y 421.014,Z 448.276,A -85,B 0,C 180,E1 -10007.603,E2 -10007.603} C_VEL
LIN {X 0,Y 420.334,Z 458.812,A -85,B 0,C 180,E1 -10008.649,E2 -10008.649} C_VEL
LIN {X 0,Y 419.701,Z 467.893,A -85,B 0,C 180,E1 -10009.757,E2 -10009.757} C_VEL
LIN {X 0,Y 419.005,Z 477.122,A -85,B 0,C 180,E1 -10011.138,E2 -10011.138} C_VEL
LIN {X 0,Y 418.413,Z 484.529,A -85,B 0,C 180,E1 -10012.508,E2 -10012.508} C_VEL
LIN {X 0,Y 418.007,Z 490.202,A -85,B 0,C 180,E1 -10013.798,E2 -10013.798} C_VEL
LIN {X 0,Y 417.633,Z 495.835,A -85,B 0,C 180,E1 -10015.411,E2 -10015.411} C_VEL
LIN {X 0,Y 417.456,Z 500.094,A -85,B 0,C 180,E1 -10017.036,E2 -10017.036} C_VEL
LIN {X 0,Y 417.176,Z 503.369,A -85,B 0,C 180,E1 -10018.833,E2 -10018.833} C_VEL
LIN {X 0,Y 417.057,Z 505.253,A -85,B 0,C 180,E1 -10020.748,E2 -10020.748} C_VEL
LIN {X 0,Y 417.042,Z 505.597,A -85,B 0,C 180,E1 -10022.633,E2 -10022.633} C_VEL
LIN {X 0,Y 417.119,Z 504.618,A -85,B 0,C 180,E1 -10024.35,E2 -10024.35} C_VEL
LIN {X 0,Y 417.295,Z 502.245,A -85,B 0,C 180,E1 -10026.118,E2 -10026.118} C_VEL
LIN {X 0,Y 417.535,Z 498.903,A -85,B 0,C 180,E1 -10027.71,E2 -10027.71} C_VEL
LIN {X 0,Y 417.878,Z 494.251,A -85,B 0,C 180,E1 -10029.317,E2 -10029.317} C_VEL
LIN {X 0,Y 418.324,Z 488.125,A -85,B 0,C 180,E1 -10030.935,E2 -10030.935} C_VEL
LIN {X 0,Y 418.874,Z 480.936,A -85,B 0,C 180,E1 -10032.417,E2 -10032.417} C_VEL
LIN {X 0,Y 419.55,Z 471.812,A -85,B 0,C 180,E1 -10033.92,E2 -10033.92} C_VEL
LIN {X 0,Y 420.28,Z 461.971,A -85,B 0,C 180,E1 -10035.211,E2 -10035.211} C_VEL
LIN {X 0,Y 421.03,Z 450.7,A -85,B 0,C 180,E1 -10036.388,E2 -10036.388} C_VEL
LIN {X 0,Y 421.72,Z 439.179,A -85,B 0,C 180,E1 -10037.336,E2 -10037.336} C_VEL
LIN {X 0,Y 422.361,Z 426.51,A -85,B 0,C 180,E1 -10038.126,E2 -10038.126} C_VEL
LIN {X 0,Y 422.467,Z 423.511,A -85,B 0,C 180,E1 -10038.285,E2 -10038.285} C_VEL
LIN {X 0,Y 419.36,Z 410.632,A -85,B 0,C 180,E1 -10038.975,E2 -10038.975} C_VEL
LIN {X 0,Y 417.429,Z 403.508,A -85,B 0,C 180,E1 -10039.283,E2 -10039.283} C_VEL
LIN {X 0,Y 417.462,Z 400.142,A -85,B 0,C 180,E1 -10042.694,E2 -10042.694} C_VEL
LIN {X 0,Y 417.627,Z 396.645,A -85,B 0,C 180,E1 -10046.266,E2 -10046.266} C_VEL
LIN {X 0,Y 417.741,Z 393.373,A -85,B 0,C 180,E1 -10049.687,E2 -10049.687} C_VEL
LIN {X 0,Y 417.84,Z 390.172,A -85,B 0,C 180,E1 -10053.054,E2 -10053.054} C_VEL
LIN {X 0,Y 417.932,Z 388.429,A -85,B 0,C 180,E1 -10055.238,E2 -10055.238} C_VEL
LIN {X 0,Y 418.208,Z 388.397,A -85,B 0,C 180,E1 -10058.302,E2 -10058.302} C_VEL
LIN {X 0,Y 418.279,Z 388.384,A -85,B 0,C 180,E1 -10061.383,E2 -10061.383} C_VEL
LIN {X 0,Y 418.297,Z 388.382,A -85,B 0,C 180,E1 -10064.406,E2 -10064.406} C_VEL
LIN {X 0,Y 418.35,Z 388.376,A -85,B 0,C 180,E1 -10067.385,E2 -10067.385} C_VEL
LIN {X 0,Y 418.337,Z 388.377,A -85,B 0,C 180,E1 -10070.328,E2 -10070.328} C_VEL
LIN {X 0,Y 418.487,Z 388.359,A -85,B 0,C 180,E1 -10073.249,E2 -10073.249} C_VEL
LIN {X 0,Y 418.335,Z 388.375,A -85,B 0,C 180,E1 -10075.181,E2 -10075.181} C_VEL
LIN {X 0,Y 418.539,Z 388.353,A -85,B 0,C 180,E1 -10078.075,E2 -10078.075} C_VEL
LIN {X 0,Y 418.666,Z 388.333,A -85,B 0,C 180,E1 -10080,E2 -10080} C_VEL
LIN {X 0,Y 418.505,Z 388.355,A -85,B 0,C 180,E1 -10082.888,E2 -10082.888} C_VEL
LIN {X 0,Y 418.487,Z 388.358,A -85,B 0,C 180,E1 -10086.751,E2 -10086.751} C_VEL
LIN {X 0,Y 418.336,Z 388.377,A -85,B 0,C 180,E1 -10089.671,E2 -10089.671} C_VEL
LIN {X 0,Y 418.341,Z 388.374,A -85,B 0,C 180,E1 -10093.001,E2 -10093.001} C_VEL
LIN {X 0,Y 418.308,Z 388.378,A -85,B 0,C 180,E1 -10096.736,E2 -10096.736} C_VEL
LIN {X 0,Y 418.266,Z 388.386,A -85,B 0,C 180,E1 -10099.79,E2 -10099.79} C_VEL
LIN {X 0,Y 418.233,Z 388.389,A -85,B 0,C 180,E1 -10102.736,E2 -10102.736} C_VEL
LIN {X 0,Y 418.267,Z 388.385,A -85,B 0,C 180,E1 -10105.904,E2 -10105.904} C_VEL
LIN {X 0,Y 418.261,Z 388.385,A -85,B 0,C 180,E1 -10109.162,E2 -10109.162} C_VEL
LIN {X 0,Y 418.253,Z 388.389,A -85,B 0,C 180,E1 -10112.844,E2 -10112.844} C_VEL
LIN {X 0,Y 418.244,Z 388.392,A -85,B 0,C 180,E1 -10116.239,E2 -10116.239} C_VEL
LIN {X 0,Y 418.263,Z 388.388,A -85,B 0,C 180,E1 -10119.681,E2 -10119.681} C_VEL
LIN {X 0,Y 418.243,Z 388.389,A -85,B 0,C 180,E1 -10122.324,E2 -10122.324} C_VEL
LIN {X 0,Y 418.234,Z 388.393,A -85,B 0,C 180,E1 -10125.109,E2 -10125.109} C_VEL
LIN {X 0,Y 418.265,Z 388.551,A -85,B 0,C 180,E1 -10126.688,E2 -10126.688} C_VEL
LIN {X 0,Y 419.29,Z 394.099,A -85,B 0,C 180,E1 -10129.811,E2 -10129.811} C_VEL
LIN {X 0,Y 420.362,Z 400.185,A -85,B 0,C 180,E1 -10132.996,E2 -10132.996} C_VEL
LIN {X 0,Y 420.35,Z 404.442,A -85,B 0,C 180,E1 -10135.01,E2 -10135.01} C_VEL
LIN {X 0,Y 419.804,Z 410.247,A -85,B 0,C 180,E1 -10137.608,E2 -10137.608} C_VEL
LIN {X 0,Y 419.226,Z 417.985,A -85,B 0,C 180,E1 -10140.912,E2 -10140.912} C_VEL
LIN {X 0,Y 418.715,Z 425.816,A -85,B 0,C 180,E1 -10144.126,E2 -10144.126} C_VEL
LIN {X 0,Y 418.288,Z 434.414,A -85,B 0,C 180,E1 -10147.534,E2 -10147.534} C_VEL
LIN {X 0,Y 417.963,Z 443.04,A -85,B 0,C 180,E1 -10150.859,E2 -10150.859} C_VEL
LIN {X 0,Y 417.719,Z 447.871,A -85,B 0,C 180,E1 -10152.684,E2 -10152.684} C_VEL
LIN {X 0,Y 420.02,Z 462.906,A -85,B 0,C 180,E1 -10153.25,E2 -10153.25} C_VEL
LIN {X 0,Y 421.79,Z 475.688,A -85,B 0,C 180,E1 -10153.918,E2 -10153.918} C_VEL
LIN {X 0,Y 421.1,Z 487.423,A -85,B 0,C 180,E1 -10154.636,E2 -10154.636} C_VEL
LIN {X 0,Y 420.385,Z 498.15,A -85,B 0,C 180,E1 -10155.477,E2 -10155.477} C_VEL
LIN {X 0,Y 419.707,Z 509.135,A -85,B 0,C 180,E1 -10156.565,E2 -10156.565} C_VEL
LIN {X 0,Y 419.126,Z 518.103,A -85,B 0,C 180,E1 -10157.655,E2 -10157.655} C_VEL
LIN {X 0,Y 418.439,Z 526.346,A -85,B 0,C 180,E1 -10158.863,E2 -10158.863} C_VEL
LIN {X 0,Y 417.913,Z 534.456,A -85,B 0,C 180,E1 -10160.319,E2 -10160.319} C_VEL
LIN {X 0,Y 417.539,Z 540.971,A -85,B 0,C 180,E1 -10161.774,E2 -10161.774} C_VEL
LIN {X 0,Y 417.271,Z 546.149,A -85,B 0,C 180,E1 -10163.229,E2 -10163.229} C_VEL
LIN {X 0,Y 417.193,Z 550.18,A -85,B 0,C 180,E1 -10164.684,E2 -10164.684} C_VEL
LIN {X 0,Y 417.036,Z 553.154,A -85,B 0,C 180,E1 -10166.135,E2 -10166.135} C_VEL
LIN {X 0,Y 417.107,Z 554.58,A -85,B 0,C 180,E1 -10167.102,E2 -10167.102} C_VEL
LIN {X 0,Y 417.035,Z 556.218,A -85,B 0,C 180,E1 -10169.034,E2 -10169.034} C_VEL
LIN {X 0,Y 417.047,Z 556.445,A -85,B 0,C 180,E1 -10170,E2 -10170} C_VEL
LIN {X 0,Y 417.035,Z 556.232,A -85,B 0,C 180,E1 -10170.965,E2 -10170.965} C_VEL
LIN {X 0,Y 417.106,Z 554.629,A -85,B 0,C 180,E1 -10172.897,E2 -10172.897} C_VEL
LIN {X 0,Y 417.035,Z 553.218,A -85,B 0,C 180,E1 -10173.865,E2 -10173.865} C_VEL
LIN {X 0,Y 417.192,Z 550.267,A -85,B 0,C 180,E1 -10175.316,E2 -10175.316} C_VEL
LIN {X 0,Y 417.275,Z 546.26,A -85,B 0,C 180,E1 -10176.77,E2 -10176.77} C_VEL
LIN {X 0,Y 417.588,Z 540.104,A -85,B 0,C 180,E1 -10178.468,E2 -10178.468} C_VEL
LIN {X 0,Y 418.015,Z 533.385,A -85,B 0,C 180,E1 -10179.923,E2 -10179.923} C_VEL
LIN {X 0,Y 418.569,Z 525.056,A -85,B 0,C 180,E1 -10181.378,E2 -10181.378} C_VEL
LIN {X 0,Y 419.257,Z 516.525,A -85,B 0,C 180,E1 -10182.586,E2 -10182.586} C_VEL
LIN {X 0,Y 419.893,Z 506.722,A -85,B 0,C 180,E1 -10183.721,E2 -10183.721} C_VEL
LIN {X 0,Y 420.554,Z 495.575,A -85,B 0,C 180,E1 -10184.764,E2 -10184.764} C_VEL
LIN {X 0,Y 421.351,Z 484.183,A -85,B 0,C 180,E1 -10185.602,E2 -10185.602} C_VEL
LIN {X 0,Y 421.777,Z 474.84,A -85,B 0,C 180,E1 -10186.144,E2 -10186.144} C_VEL
LIN {X 0,Y 419.901,Z 461.793,A -85,B 0,C 180,E1 -10186.806,E2 -10186.806} C_VEL
LIN {X 0,Y 417.738,Z 448.428,A -85,B 0,C 180,E1 -10187.286,E2 -10187.286} C_VEL
LIN {X 0,Y 418.155,Z 439.582,A -85,B 0,C 180,E1 -10190.667,E2 -10190.667} C_VEL
LIN {X 0,Y 418.583,Z 430.342,A -85,B 0,C 180,E1 -10194.289,E2 -10194.289} C_VEL
LIN {X 0,Y 418.997,Z 422.999,A -85,B 0,C 180,E1 -10197.253,E2 -10197.253} C_VEL
LIN {X 0,Y 419.447,Z 415.955,A -85,B 0,C 180,E1 -10200.175,E2 -10200.175} C_VEL
LIN {X 0,Y 420.104,Z 408.167,A -85,B 0,C 180,E1 -10203.508,E2 -10203.508} C_VEL
LIN {X 0,Y 420.531,Z 403.025,A -85,B 0,C 180,E1 -10205.797,E2 -10205.797} C_VEL
LIN {X 0,Y 420.238,Z 399.27,A -85,B 0,C 180,E1 -10207.569,E2 -10207.569} C_VEL
LIN {X 0,Y 419.07,Z 392.77,A -85,B 0,C 180,E1 -10210.846,E2 -10210.846} C_VEL
LIN {X 0,Y 418.229,Z 388.391,A -85,B 0,C 180,E1 -10213.226,E2 -10213.226} C_VEL
LIN {X 0,Y 418.204,Z 388.394,A -85,B 0,C 180,E1 -10216.448,E2 -10216.448} C_VEL
LIN {X 0,Y 418.26,Z 388.387,A -85,B 0,C 180,E1 -10219.123,E2 -10219.123} C_VEL
LIN {X 0,Y 418.233,Z 388.389,A -85,B 0,C 180,E1 -10222.164,E2 -10222.164} C_VEL
LIN {X 0,Y 418.259,Z 388.386,A -85,B 0,C 180,E1 -10225.419,E2 -10225.419} C_VEL
LIN {X 0,Y 418.205,Z 388.393,A -85,B 0,C 180,E1 -10228.603,E2 -10228.603} C_VEL
LIN {X 0,Y 418.284,Z 388.381,A -85,B 0,C 180,E1 -10231.936,E2 -10231.936} C_VEL
LIN {X 0,Y 418.282,Z 388.383,A -85,B 0,C 180,E1 -10235.162,E2 -10235.162} C_VEL
LIN {X 0,Y 418.226,Z 388.389,A -85,B 0,C 180,E1 -10238.303,E2 -10238.303} C_VEL
LIN {X 0,Y 418.275,Z 388.383,A -85,B 0,C 180,E1 -10241.383,E2 -10241.383} C_VEL
LIN {X 0,Y 418.293,Z 388.383,A -85,B 0,C 180,E1 -10244.406,E2 -10244.406} C_VEL
LIN {X 0,Y 418.346,Z 388.373,A -85,B 0,C 180,E1 -10247.385,E2 -10247.385} C_VEL
LIN {X 0,Y 418.333,Z 388.377,A -85,B 0,C 180,E1 -10250.329,E2 -10250.329} C_VEL
LIN {X 0,Y 418.483,Z 388.357,A -85,B 0,C 180,E1 -10253.249,E2 -10253.249} C_VEL
LIN {X 0,Y 418.332,Z 388.376,A -85,B 0,C 180,E1 -10255.182,E2 -10255.182} C_VEL
LIN {X 0,Y 418.536,Z 388.35,A -85,B 0,C 180,E1 -10258.076,E2 -10258.076} C_VEL
LIN {X 0,Y 418.665,Z 388.334,A -85,B 0,C 180,E1 -10260,E2 -10260} C_VEL
LIN {X 0,Y 418.503,Z 388.356,A -85,B 0,C 180,E1 -10262.888,E2 -10262.888} C_VEL
LIN {X 0,Y 418.485,Z 388.359,A -85,B 0,C 180,E1 -10266.751,E2 -10266.751} C_VEL
LIN {X 0,Y 418.392,Z 388.37,A -85,B 0,C 180,E1 -10268.695,E2 -10268.695} C_VEL
LIN {X 0,Y 418.309,Z 388.378,A -85,B 0,C 180,E1 -10271.631,E2 -10271.631} C_VEL
LIN {X 0,Y 418.294,Z 388.383,A -85,B 0,C 180,E1 -10274.597,E2 -10274.597} C_VEL
LIN {X 0,Y 418.28,Z 388.381,A -85,B 0,C 180,E1 -10277.604,E2 -10277.604} C_VEL
LIN {X 0,Y 418.242,Z 388.389,A -85,B 0,C 180,E1 -10280.664,E2 -10280.664} C_VEL
LIN {X 0,Y 418.281,Z 388.382,A -85,B 0,C 180,E1 -10283.782,E2 -10283.782} C_VEL
LIN {X 0,Y 418.303,Z 388.379,A -85,B 0,C 180,E1 -10287.071,E2 -10287.071} C_VEL
LIN {X 0,Y 418.238,Z 388.39,A -85,B 0,C 180,E1 -10290.273,E2 -10290.273} C_VEL
LIN {X 0,Y 418.243,Z 388.387,A -85,B 0,C 180,E1 -10293.678,E2 -10293.678} C_VEL
LIN {X 0,Y 418.243,Z 388.386,A -85,B 0,C 180,E1 -10297.224,E2 -10297.224} C_VEL
LIN {X 0,Y 418.261,Z 388.385,A -85,B 0,C 180,E1 -10299.681,E2 -10299.681} C_VEL
LIN {X 0,Y 418.241,Z 388.39,A -85,B 0,C 180,E1 -10302.325,E2 -10302.325} C_VEL
LIN {X 0,Y 418.232,Z 388.387,A -85,B 0,C 180,E1 -10305.11,E2 -10305.11} C_VEL
LIN {X 0,Y 418.237,Z 388.389,A -85,B 0,C 180,E1 -10307.768,E2 -10307.768} C_VEL
LIN {X 0,Y 418.258,Z 388.385,A -85,B 0,C 180,E1 -10310.619,E2 -10310.619} C_VEL
LIN {X 0,Y 418.244,Z 388.389,A -85,B 0,C 180,E1 -10313.977,E2 -10313.977} C_VEL
LIN {X 0,Y 418.257,Z 388.384,A -85,B 0,C 180,E1 -10317.157,E2 -10317.157} C_VEL
LIN {X 0,Y 418.269,Z 388.382,A -85,B 0,C 180,E1 -10320.896,E2 -10320.896} C_VEL
LIN {X 0,Y 418.272,Z 388.386,A -85,B 0,C 180,E1 -10324.097,E2 -10324.097} C_VEL
LIN {X 0,Y 418.24,Z 388.387,A -85,B 0,C 180,E1 -10327.265,E2 -10327.265} C_VEL
LIN {X 0,Y 418.285,Z 388.382,A -85,B 0,C 180,E1 -10330.365,E2 -10330.365} C_VEL
LIN {X 0,Y 418.32,Z 388.378,A -85,B 0,C 180,E1 -10333.405,E2 -10333.405} C_VEL
LIN {X 0,Y 418.349,Z 388.373,A -85,B 0,C 180,E1 -10337,E2 -10337} C_VEL
LIN {X 0,Y 418.343,Z 388.374,A -85,B 0,C 180,E1 -10340.329,E2 -10340.329} C_VEL
LIN {X 0,Y 418.517,Z 388.353,A -85,B 0,C 180,E1 -10342.28,E2 -10342.28} C_VEL
LIN {X 0,Y 418.517,Z 388.354,A -85,B 0,C 180,E1 -10344.218,E2 -10344.218} C_VEL
LIN {X 0,Y 418.47,Z 388.362,A -85,B 0,C 180,E1 -10348.075,E2 -10348.075} C_VEL
LIN {X 0,Y 418.217,Z 388.393,A -85,B 0,C 180,E1 -10350,E2 -10350} C_VEL
LIN {X 0,Y 417.76,Z 388.452,A -85,B 0,C 180,E1 -10350.964,E2 -10350.964} C_VEL
LIN {X 0,Y 417.778,Z 391.163,A -85,B 0,C 180,E1 -10353.858,E2 -10353.858} C_VEL
LIN {X 0,Y 417.709,Z 394.258,A -85,B 0,C 180,E1 -10356.933,E2 -10356.933} C_VEL
LIN {X 0,Y 417.483,Z 398.062,A -85,B 0,C 180,E1 -10360.671,E2 -10360.671} C_VEL
LIN {X 0,Y 417.424,Z 400.714,A -85,B 0,C 180,E1 -10363.197,E2 -10363.197} C_VEL
LIN {X 0,Y 417.324,Z 401.912,A -85,B 0,C 180,E1 -10363.689,E2 -10363.689} C_VEL
LIN {X 0,Y 417.117,Z 404.072,A -85,B 0,C 180,E1 -10364.12,E2 -10364.12} C_VEL
LIN {X 0,Y 416.691,Z 408.454,A -85,B 0,C 180,E1 -10364.651,E2 -10364.651} C_VEL
LIN {X 0,Y 416.195,Z 413.824,A -85,B 0,C 180,E1 -10365.07,E2 -10365.07} C_VEL
LIN {X 0,Y 415.437,Z 425.566,A -85,B 0,C 180,E1 -10365.74,E2 -10365.74} C_VEL
LIN {X 0,Y 414.798,Z 437.651,A -85,B 0,C 180,E1 -10366.487,E2 -10366.487} C_VEL
LIN {X 0,Y 414.124,Z 449.08,A -85,B 0,C 180,E1 -10367.404,E2 -10367.404} C_VEL
LIN {X 0,Y 413.413,Z 459.583,A -85,B 0,C 180,E1 -10368.472,E2 -10368.472} C_VEL
LIN {X 0,Y 412.706,Z 469.008,A -85,B 0,C 180,E1 -10369.653,E2 -10369.653} C_VEL
LIN {X 0,Y 412.025,Z 477.715,A -85,B 0,C 180,E1 -10370.99,E2 -10370.99} C_VEL
LIN {X 0,Y 411.417,Z 485.015,A -85,B 0,C 180,E1 -10372.367,E2 -10372.367} C_VEL
LIN {X 0,Y 410.912,Z 491.755,A -85,B 0,C 180,E1 -10373.966,E2 -10373.966} C_VEL
LIN {X 0,Y 410.593,Z 496.347,A -85,B 0,C 180,E1 -10375.335,E2 -10375.335} C_VEL
LIN {X 0,Y 410.38,Z 500.744,A -85,B 0,C 180,E1 -10377.059,E2 -10377.059} C_VEL
LIN {X 0,Y 410.074,Z 504.17,A -85,B 0,C 180,E1 -10379.066,E2 -10379.066} C_VEL
LIN {X 0,Y 409.957,Z 505.823,A -85,B 0,C 180,E1 -10381,E2 -10381} C_VEL
LIN {X 0,Y 409.968,Z 505.998,A -85,B 0,C 180,E1 -10382.86,E2 -10382.86} C_VEL
LIN {X 0,Y 410.044,Z 504.796,A -85,B 0,C 180,E1 -10384.643,E2 -10384.643} C_VEL
LIN {X 0,Y 410.274,Z 502.358,A -85,B 0,C 180,E1 -10386.378,E2 -10386.378} C_VEL
LIN {X 0,Y 410.546,Z 498.759,A -85,B 0,C 180,E1 -10388.051,E2 -10388.051} C_VEL
LIN {X 0,Y 410.9,Z 493.97,A -85,B 0,C 180,E1 -10389.675,E2 -10389.675} C_VEL
LIN {X 0,Y 411.366,Z 487.849,A -85,B 0,C 180,E1 -10391.26,E2 -10391.26} C_VEL
LIN {X 0,Y 411.98,Z 480.23,A -85,B 0,C 180,E1 -10392.816,E2 -10392.816} C_VEL
LIN {X 0,Y 412.719,Z 471.258,A -85,B 0,C 180,E1 -10394.279,E2 -10394.279} C_VEL
LIN {X 0,Y 413.45,Z 461.451,A -85,B 0,C 180,E1 -10395.555,E2 -10395.555} C_VEL
LIN {X 0,Y 414.224,Z 450.499,A -85,B 0,C 180,E1 -10396.7,E2 -10396.7} C_VEL
LIN {X 0,Y 414.935,Z 439.3,A -85,B 0,C 180,E1 -10397.623,E2 -10397.623} C_VEL
LIN {X 0,Y 415.546,Z 427.63,A -85,B 0,C 180,E1 -10398.367,E2 -10398.367} C_VEL
LIN {X 0,Y 415.451,Z 423.78,A -85,B 0,C 180,E1 -10398.585,E2 -10398.585} C_VEL
LIN {X 0,Y 412.286,Z 410.947,A -85,B 0,C 180,E1 -10399.289,E2 -10399.289} C_VEL
LIN {X 0,Y 410.382,Z 403.956,A -85,B 0,C 180,E1 -10399.608,E2 -10399.608} C_VEL
LIN {X 0,Y 410.439,Z 400.066,A -85,B 0,C 180,E1 -10403.589,E2 -10403.589} C_VEL
LIN {X 0,Y 410.631,Z 396.787,A -85,B 0,C 180,E1 -10406.996,E2 -10406.996} C_VEL
LIN {X 0,Y 410.704,Z 393.726,A -85,B 0,C 180,E1 -10410.247,E2 -10410.247} C_VEL
LIN {X 0,Y 410.793,Z 390.6,A -85,B 0,C 180,E1 -10413.588,E2 -10413.588} C_VEL
LIN {X 0,Y 410.862,Z 389.31,A -85,B 0,C 180,E1 -10415.037,E2 -10415.037} C_VEL
LIN {X 0,Y 411.163,Z 389.275,A -85,B 0,C 180,E1 -10417.911,E2 -10417.911} C_VEL
LIN {X 0,Y 411.22,Z 389.265,A -85,B 0,C 180,E1 -10421.051,E2 -10421.051} C_VEL
LIN {X 0,Y 411.249,Z 389.259,A -85,B 0,C 180,E1 -10424.131,E2 -10424.131} C_VEL
LIN {X 0,Y 411.298,Z 389.255,A -85,B 0,C 180,E1 -10427.165,E2 -10427.165} C_VEL
LIN {X 0,Y 411.289,Z 389.254,A -85,B 0,C 180,E1 -10430.161,E2 -10430.161} C_VEL
LIN {X 0,Y 411.451,Z 389.235,A -85,B 0,C 180,E1 -10433.133,E2 -10433.133} C_VEL
LIN {X 0,Y 411.306,Z 389.25,A -85,B 0,C 180,E1 -10435.099,E2 -10435.099} C_VEL
LIN {X 0,Y 411.508,Z 389.228,A -85,B 0,C 180,E1 -10438.042,E2 -10438.042} C_VEL
LIN {X 0,Y 411.636,Z 389.209,A -85,B 0,C 180,E1 -10440,E2 -10440} C_VEL
LIN {X 0,Y 411.46,Z 389.233,A -85,B 0,C 180,E1 -10442.937,E2 -10442.937} C_VEL
LIN {X 0,Y 411.45,Z 389.234,A -85,B 0,C 180,E1 -10446.867,E2 -10446.867} C_VEL
LIN {X 0,Y 411.288,Z 389.256,A -85,B 0,C 180,E1 -10449.839,E2 -10449.839} C_VEL
LIN {X 0,Y 411.3,Z 389.251,A -85,B 0,C 180,E1 -10453.104,E2 -10453.104} C_VEL
LIN {X 0,Y 411.252,Z 389.257,A -85,B 0,C 180,E1 -10456.889,E2 -10456.889} C_VEL
LIN {X 0,Y 411.226,Z 389.263,A -85,B 0,C 180,E1 -10459.987,E2 -10459.987} C_VEL
LIN {X 0,Y 411.198,Z 389.267,A -85,B 0,C 180,E1 -10463.148,E2 -10463.148} C_VEL
LIN {X 0,Y 411.234,Z 389.259,A -85,B 0,C 180,E1 -10466.381,E2 -10466.381} C_VEL
LIN {X 0,Y 411.196,Z 389.268,A -85,B 0,C 180,E1 -10469.713,E2 -10469.713} C_VEL
LIN {X 0,Y 411.202,Z 389.267,A -85,B 0,C 180,E1 -10473.156,E2 -10473.156} C_VEL
LIN {X 0,Y 411.192,Z 389.27,A -85,B 0,C 180,E1 -10476.553,E2 -10476.553} C_VEL
LIN {X 0,Y 411.225,Z 389.265,A -85,B 0,C 180,E1 -10479.731,E2 -10479.731} C_VEL
LIN {X 0,Y 411.175,Z 389.268,A -85,B 0,C 180,E1 -10483.133,E2 -10483.133} C_VEL
LIN {X 0,Y 411.169,Z 389.346,A -85,B 0,C 180,E1 -10486.223,E2 -10486.223} C_VEL
LIN {X 0,Y 411.99,Z 393.436,A -85,B 0,C 180,E1 -10488.641,E2 -10488.641} C_VEL
LIN {X 0,Y 413.156,Z 400.011,A -85,B 0,C 180,E1 -10492.239,E2 -10492.239} C_VEL
LIN {X 0,Y 413.488,Z 403.754,A -85,B 0,C 180,E1 -10494.099,E2 -10494.099} C_VEL
LIN {X 0,Y 412.923,Z 410.032,A -85,B 0,C 180,E1 -10497,E2 -10497} C_VEL
LIN {X 0,Y 412.283,Z 417.749,A -85,B 0,C 180,E1 -10500.386,E2 -10500.386} C_VEL
LIN {X 0,Y 411.76,Z 425.515,A -85,B 0,C 180,E1 -10503.655,E2 -10503.655} C_VEL
LIN {X 0,Y 411.23,Z 434.599,A -85,B 0,C 180,E1 -10507.35,E2 -10507.35} C_VEL
LIN {X 0,Y 410.865,Z 443.964,A -85,B 0,C 180,E1 -10511.034,E2 -10511.034} C_VEL
LIN {X 0,Y 410.686,Z 447.702,A -85,B 0,C 180,E1 -10512.402,E2 -10512.402} C_VEL
LIN {X 0,Y 412.799,Z 461.043,A -85,B 0,C 180,E1 -10512.891,E2 -10512.891} C_VEL
LIN {X 0,Y 414.639,Z 474.127,A -85,B 0,C 180,E1 -10513.57,E2 -10513.57} C_VEL
LIN {X 0,Y 414.781,Z 478.552,A -85,B 0,C 180,E1 -10513.829,E2 -10513.829} C_VEL
LIN {X 0,Y 413.989,Z 490.28,A -85,B 0,C 180,E1 -10514.618,E2 -10514.618} C_VEL
LIN {X 0,Y 413.233,Z 501.539,A -85,B 0,C 180,E1 -10515.588,E2 -10515.588} C_VEL
LIN {X 0,Y 412.532,Z 511.907,A -85,B 0,C 180,E1 -10516.704,E2 -10516.704} C_VEL
LIN {X 0,Y 411.831,Z 521.155,A -85,B 0,C 180,E1 -10517.933,E2 -10517.933} C_VEL
LIN {X 0,Y 411.123,Z 530.175,A -85,B 0,C 180,E1 -10519.411,E2 -10519.411} C_VEL
LIN {X 0,Y 410.679,Z 537.455,A -85,B 0,C 180,E1 -10520.892,E2 -10520.892} C_VEL
LIN {X 0,Y 410.354,Z 542.371,A -85,B 0,C 180,E1 -10522.125,E2 -10522.125} C_VEL
LIN {X 0,Y 410.173,Z 547.177,A -85,B 0,C 180,E1 -10523.611,E2 -10523.611} C_VEL
LIN {X 0,Y 410.096,Z 550.83,A -85,B 0,C 180,E1 -10525.084,E2 -10525.084} C_VEL
LIN {X 0,Y 409.955,Z 552.718,A -85,B 0,C 180,E1 -10526.068,E2 -10526.068} C_VEL
LIN {X 0,Y 410.007,Z 554.146,A -85,B 0,C 180,E1 -10527.052,E2 -10527.052} C_VEL
LIN {X 0,Y 409.988,Z 555.164,A -85,B 0,C 180,E1 -10528.035,E2 -10528.035} C_VEL
LIN {X 0,Y 409.959,Z 555.788,A -85,B 0,C 180,E1 -10529.017,E2 -10529.017} C_VEL
LIN {X 0,Y 409.967,Z 556.016,A -85,B 0,C 180,E1 -10530,E2 -10530} C_VEL
LIN {X 0,Y 409.959,Z 555.805,A -85,B 0,C 180,E1 -10530.982,E2 -10530.982} C_VEL
LIN {X 0,Y 409.988,Z 555.201,A -85,B 0,C 180,E1 -10531.964,E2 -10531.964} C_VEL
LIN {X 0,Y 410.007,Z 554.202,A -85,B 0,C 180,E1 -10532.947,E2 -10532.947} C_VEL
LIN {X 0,Y 409.954,Z 552.792,A -85,B 0,C 180,E1 -10533.932,E2 -10533.932} C_VEL
LIN {X 0,Y 410.107,Z 549.84,A -85,B 0,C 180,E1 -10535.408,E2 -10535.408} C_VEL
LIN {X 0,Y 410.197,Z 545.833,A -85,B 0,C 180,E1 -10536.888,E2 -10536.888} C_VEL
LIN {X 0,Y 410.55,Z 539.675,A -85,B 0,C 180,E1 -10538.614,E2 -10538.614} C_VEL
LIN {X 0,Y 410.993,Z 532.953,A -85,B 0,C 180,E1 -10540.094,E2 -10540.094} C_VEL
LIN {X 0,Y 411.575,Z 524.618,A -85,B 0,C 180,E1 -10541.574,E2 -10541.574} C_VEL
LIN {X 0,Y 412.257,Z 516.077,A -85,B 0,C 180,E1 -10542.804,E2 -10542.804} C_VEL
LIN {X 0,Y 413.007,Z 505.077,A -85,B 0,C 180,E1 -10544.081,E2 -10544.081} C_VEL
LIN {X 0,Y 413.796,Z 493.681,A -85,B 0,C 180,E1 -10545.137,E2 -10545.137} C_VEL
LIN {X 0,Y 414.624,Z 481.771,A -85,B 0,C 180,E1 -10545.988,E2 -10545.988} C_VEL
LIN {X 0,Y 414.842,Z 475.488,A -85,B 0,C 180,E1 -10546.358,E2 -10546.358} C_VEL
LIN {X 0,Y 412.957,Z 462.154,A -85,B 0,C 180,E1 -10547.064,E2 -10547.064} C_VEL
LIN {X 0,Y 410.71,Z 447.981,A -85,B 0,C 180,E1 -10547.602,E2 -10547.602} C_VEL
LIN {X 0,Y 411.095,Z 439.207,A -85,B 0,C 180,E1 -10551.039,E2 -10551.039} C_VEL
LIN {X 0,Y 411.492,Z 431.33,A -85,B 0,C 180,E1 -10554.198,E2 -10554.198} C_VEL
LIN {X 0,Y 411.967,Z 423.469,A -85,B 0,C 180,E1 -10557.426,E2 -10557.426} C_VEL
LIN {X 0,Y 412.528,Z 415.687,A -85,B 0,C 180,E1 -10560.736,E2 -10560.736} C_VEL
LIN {X 0,Y 413.22,Z 407.925,A -85,B 0,C 180,E1 -10564.142,E2 -10564.142} C_VEL
LIN {X 0,Y 413.52,Z 402.796,A -85,B 0,C 180,E1 -10566.5,E2 -10566.5} C_VEL
LIN {X 0,Y 412.751,Z 397.656,A -85,B 0,C 180,E1 -10569.049,E2 -10569.049} C_VEL
LIN {X 0,Y 411.82,Z 392.548,A -85,B 0,C 180,E1 -10571.724,E2 -10571.724} C_VEL
LIN {X 0,Y 411.173,Z 389.27,A -85,B 0,C 180,E1 -10573.594,E2 -10573.594} C_VEL
LIN {X 0,Y 411.172,Z 389.269,A -85,B 0,C 180,E1 -10576.866,E2 -10576.866} C_VEL
LIN {X 0,Y 411.222,Z 389.263,A -85,B 0,C 180,E1 -10580.269,E2 -10580.269} C_VEL
LIN {X 0,Y 411.19,Z 389.266,A -85,B 0,C 180,E1 -10583.446,E2 -10583.446} C_VEL
